LIN {X 0,Y 573.228,Z 217.081,A -85,B 0,C 180,E1 -2311.435,E2 -2311.435} C_VEL
LIN {X 0,Y 573.254,Z 217.075,A -85,B 0,C 180,E1 -2314.59,E2 -2314.59} C_VEL
LIN {X 0,Y 573.238,Z 217.078,A -85,B 0,C 180,E1 -2317.662,E2 -2317.662} C_VEL
LIN {X 0,Y 573.273,Z 217.079,A -85,B 0,C 180,E1 -2320.67,E2 -2320.67} C_VEL
LIN {X 0,Y 573.21,Z 217.081,A -85,B 0,C 180,E1 -2323.621,E2 -2323.621} C_VEL
LIN {X 0,Y 573.252,Z 217.08,A -85,B 0,C 180,E1 -2325.807,E2 -2325.807} C_VEL
LIN {X 0,Y 573.232,Z 217.077,A -85,B 0,C 180,E1 -2328.765,E2 -2328.765} C_VEL
LIN {X 0,Y 573.248,Z 217.08,A -85,B 0,C 180,E1 -2331.54,E2 -2331.54} C_VEL
LIN {X 0,Y 573.243,Z 217.077,A -85,B 0,C 180,E1 -2333.665,E2 -2333.665} C_VEL
LIN {X 0,Y 573.225,Z 217.079,A -85,B 0,C 180,E1 -2335.781,E2 -2335.781} C_VEL
LIN {X 0,Y 573.311,Z 217.07,A -85,B 0,C 180,E1 -2337.892,E2 -2337.892} C_VEL
LIN {X 0,Y 573.326,Z 217.067,A -85,B 0,C 180,E1 -2340.702,E2 -2340.702} C_VEL
LIN {X 0,Y 573.292,Z 217.07,A -85,B 0,C 180,E1 -2342.811,E2 -2342.811} C_VEL
LIN {X 0,Y 573.274,Z 217.077,A -85,B 0,C 180,E1 -2345.628,E2 -2345.628} C_VEL
LIN {X 0,Y 573.235,Z 217.078,A -85,B 0,C 180,E1 -2348.46,E2 -2348.46} C_VEL
LIN {X 0,Y 573.28,Z 217.073,A -85,B 0,C 180,E1 -2351.312,E2 -2351.312} C_VEL
LIN {X 0,Y 573.283,Z 217.078,A -85,B 0,C 180,E1 -2354.422,E2 -2354.422} C_VEL
LIN {X 0,Y 573.266,Z 217.074,A -85,B 0,C 180,E1 -2357.112,E2 -2357.112} C_VEL
LIN {X 0,Y 573.244,Z 217.078,A -85,B 0,C 180,E1 -2360.077,E2 -2360.077} C_VEL
LIN {X 0,Y 573.227,Z 217.078,A -85,B 0,C 180,E1 -2362.338,E2 -2362.338} C_VEL
LIN {X 0,Y 573.193,Z 217.083,A -85,B 0,C 180,E1 -2364.335,E2 -2364.335} C_VEL
LIN {X 0,Y 572.549,Z 217.17,A -85,B 0,C 180,E1 -2364.921,E2 -2364.921} C_VEL
LIN {X 0,Y 569.716,Z 217.52,A -85,B 0,C 180,E1 -2365.873,E2 -2365.873} C_VEL
LIN {X 0,Y 567.301,Z 217.822,A -85,B 0,C 180,E1 -2366.638,E2 -2366.638} C_VEL
LIN {X 0,Y 566.251,Z 217.949,A -85,B 0,C 180,E1 -2367.229,E2 -2367.229} C_VEL
LIN {X 0,Y 566.158,Z 217.958,A -85,B 0,C 180,E1 -2367.43,E2 -2367.43} C_VEL
LIN {X 0,Y 566.175,Z 217.958,A -85,B 0,C 180,E1 -2369.771,E2 -2369.771} C_VEL
LIN {X 0,Y 566.209,Z 217.956,A -85,B 0,C 180,E1 -2372.429,E2 -2372.429} C_VEL
LIN {X 0,Y 566.186,Z 217.956,A -85,B 0,C 180,E1 -2374.989,E2 -2374.989} C_VEL
LIN {X 0,Y 566.199,Z 217.96,A -85,B 0,C 180,E1 -2377.461,E2 -2377.461} C_VEL
LIN {X 0,Y 566.214,Z 217.952,A -85,B 0,C 180,E1 -2380.199,E2 -2380.199} C_VEL
LIN {X 0,Y 566.193,Z 217.958,A -85,B 0,C 180,E1 -2383.055,E2 -2383.055} C_VEL
LIN {X 0,Y 566.15,Z 217.964,A -85,B 0,C 180,E1 -2386.054,E2 -2386.054} C_VEL
LIN {X 0,Y 566.141,Z 217.96,A -85,B 0,C 180,E1 -2388.856,E2 -2388.856} C_VEL
LIN {X 0,Y 566.187,Z 217.963,A -85,B 0,C 180,E1 -2391.636,E2 -2391.636} C_VEL
LIN {X 0,Y 566.158,Z 217.959,A -85,B 0,C 180,E1 -2394.307,E2 -2394.307} C_VEL
LIN {X 0,Y 566.206,Z 217.959,A -85,B 0,C 180,E1 -2396.896,E2 -2396.896} C_VEL
LIN {X 0,Y 566.063,Z 217.978,A -85,B 0,C 180,E1 -2399.399,E2 -2399.399} C_VEL
LIN {X 0,Y 566.018,Z 219.482,A -85,B 0,C 180,E1 -2401.036,E2 -2401.036} C_VEL
LIN {X 0,Y 565.984,Z 222.214,A -85,B 0,C 180,E1 -2403.446,E2 -2403.446} C_VEL
LIN {X 0,Y 565.96,Z 224.896,A -85,B 0,C 180,E1 -2405.807,E2 -2405.807} C_VEL
LIN {X 0,Y 565.943,Z 228.388,A -85,B 0,C 180,E1 -2408.891,E2 -2408.891} C_VEL
LIN {X 0,Y 565.917,Z 230.996,A -85,B 0,C 180,E1 -2411.161,E2 -2411.161} C_VEL
LIN {X 0,Y 565.897,Z 233.568,A -85,B 0,C 180,E1 -2413.402,E2 -2413.402} C_VEL
LIN {X 0,Y 565.876,Z 237.059,A -85,B 0,C 180,E1 -2416.35,E2 -2416.35} C_VEL
LIN {X 0,Y 565.887,Z 240.835,A -85,B 0,C 180,E1 -2419.263,E2 -2419.263} C_VEL
LIN {X 0,Y 565.847,Z 243.676,A -85,B 0,C 180,E1 -2421.427,E2 -2421.427} C_VEL
LIN {X 0,Y 566.921,Z 251.031,A -85,B 0,C 180,E1 -2421.623,E2 -2421.623} C_VEL
LIN {X 0,Y 566.792,Z 264.125,A -85,B 0,C 180,E1 -2422.025,E2 -2422.025} C_VEL
LIN {X 0,Y 566.713,Z 275.551,A -85,B 0,C 180,E1 -2422.517,E2 -2422.517} C_VEL
LIN {X 0,Y 566.463,Z 287.212,A -85,B 0,C 180,E1 -2423.168,E2 -2423.168} C_VEL
LIN {X 0,Y 566.41,Z 298.182,A -85,B 0,C 180,E1 -2423.945,E2 -2423.945} C_VEL
LIN {X 0,Y 566.23,Z 308.312,A -85,B 0,C 180,E1 -2424.836,E2 -2424.836} C_VEL
LIN {X 0,Y 566.159,Z 316.567,A -85,B 0,C 180,E1 -2425.728,E2 -2425.728} C_VEL
LIN {X 0,Y 566.083,Z 324.665,A -85,B 0,C 180,E1 -2426.796,E2 -2426.796} C_VEL
LIN {X 0,Y 565.912,Z 331.198,A -85,B 0,C 180,E1 -2427.864,E2 -2427.864} C_VEL
LIN {X 0,Y 565.961,Z 336.406,A -85,B 0,C 180,E1 -2428.932,E2 -2428.932} C_VEL
LIN {X 0,Y 565.872,Z 340.467,A -85,B 0,C 180,E1 -2429.999,E2 -2429.999} C_VEL
LIN {X 0,Y 565.846,Z 342.6,A -85,B 0,C 180,E1 -2430.711,E2 -2430.711} C_VEL
LIN {X 0,Y 565.847,Z 344.276,A -85,B 0,C 180,E1 -2431.422,E2 -2431.422} C_VEL
LIN {X 0,Y 565.873,Z 346.433,A -85,B 0,C 180,E1 -2432.847,E2 -2432.847} C_VEL
LIN {X 0,Y 565.911,Z 346.898,A -85,B 0,C 180,E1 -2433.559,E2 -2433.559} C_VEL
LIN {X 0,Y 565.911,Z 346.957,A -85,B 0,C 180,E1 -2434.272,E2 -2434.272} C_VEL
LIN {X 0,Y 565.898,Z 345.923,A -85,B 0,C 180,E1 -2435.701,E2 -2435.701} C_VEL
LIN {X 0,Y 565.918,Z 344.547,A -85,B 0,C 180,E1 -2436.533,E2 -2436.533} C_VEL
LIN {X 0,Y 565.902,Z 341.227,A -85,B 0,C 180,E1 -2437.851,E2 -2437.851} C_VEL
LIN {X 0,Y 565.93,Z 337.36,A -85,B 0,C 180,E1 -2438.929,E2 -2438.929} C_VEL
LIN {X 0,Y 565.978,Z 332.342,A -85,B 0,C 180,E1 -2440.01,E2 -2440.01} C_VEL
LIN {X 0,Y 566.048,Z 325.124,A -85,B 0,C 180,E1 -2441.227,E2 -2441.227} C_VEL
LIN {X 0,Y 566.158,Z 316.558,A -85,B 0,C 180,E1 -2442.364,E2 -2442.364} C_VEL
LIN {X 0,Y 566.247,Z 308.118,A -85,B 0,C 180,E1 -2443.273,E2 -2443.273} C_VEL
LIN {X 0,Y 566.372,Z 297.678,A -85,B 0,C 180,E1 -2444.185,E2 -2444.185} C_VEL
LIN {X 0,Y 566.493,Z 286.979,A -85,B 0,C 180,E1 -2444.936,E2 -2444.936} C_VEL
LIN {X 0,Y 566.655,Z 275.898,A -85,B 0,C 180,E1 -2445.556,E2 -2445.556} C_VEL
LIN {X 0,Y 566.771,Z 264.256,A -85,B 0,C 180,E1 -2446.061,E2 -2446.061} C_VEL
LIN {X 0,Y 566.882,Z 250.786,A -85,B 0,C 180,E1 -2446.474,E2 -2446.474} C_VEL
LIN {X 0,Y 565.905,Z 243.69,A -85,B 0,C 180,E1 -2446.651,E2 -2446.651} C_VEL
LIN {X 0,Y 565.849,Z 239.839,A -85,B 0,C 180,E1 -2449.592,E2 -2449.592} C_VEL
LIN {X 0,Y 565.836,Z 236.886,A -85,B 0,C 180,E1 -2451.876,E2 -2451.876} C_VEL
LIN {X 0,Y 565.892,Z 234.162,A -85,B 0,C 180,E1 -2454.193,E2 -2454.193} C_VEL
LIN {X 0,Y 565.953,Z 231.389,A -85,B 0,C 180,E1 -2456.607,E2 -2456.607} C_VEL
LIN {X 0,Y 566.002,Z 227.922,A -85,B 0,C 180,E1 -2459.635,E2 -2459.635} C_VEL
LIN {X 0,Y 566.007,Z 224.804,A -85,B 0,C 180,E1 -2462.398,E2 -2462.398} C_VEL
LIN {X 0,Y 566.02,Z 221.892,A -85,B 0,C 180,E1 -2464.966,E2 -2464.966} C_VEL
LIN {X 0,Y 566.031,Z 219.071,A -85,B 0,C 180,E1 -2467.472,E2 -2467.472} C_VEL
LIN {X 0,Y 566.035,Z 217.981,A -85,B 0,C 180,E1 -2468.535,E2 -2468.535} C_VEL
LIN {X 0,Y 566.202,Z 217.957,A -85,B 0,C 180,E1 -2470.785,E2 -2470.785} C_VEL
LIN {X 0,Y 566.196,Z 217.957,A -85,B 0,C 180,E1 -2473.053,E2 -2473.053} C_VEL
LIN {X 0,Y 566.187,Z 217.962,A -85,B 0,C 180,E1 -2476.048,E2 -2476.048} C_VEL
LIN {X 0,Y 566.195,Z 217.961,A -85,B 0,C 180,E1 -2479.214,E2 -2479.214} C_VEL
LIN {X 0,Y 566.181,Z 217.957,A -85,B 0,C 180,E1 -2481.636,E2 -2481.636} C_VEL
LIN {X 0,Y 566.205,Z 217.96,A -85,B 0,C 180,E1 -2484.311,E2 -2484.311} C_VEL
LIN {X 0,Y 566.195,Z 217.955,A -85,B 0,C 180,E1 -2486.896,E2 -2486.896} C_VEL
LIN {X 0,Y 566.162,Z 217.963,A -85,B 0,C 180,E1 -2489.406,E2 -2489.406} C_VEL
LIN {X 0,Y 566.219,Z 217.952,A -85,B 0,C 180,E1 -2491.858,E2 -2491.858} C_VEL
LIN {X 0,Y 566.217,Z 217.957,A -85,B 0,C 180,E1 -2494.251,E2 -2494.251} C_VEL
LIN {X 0,Y 566.181,Z 217.957,A -85,B 0,C 180,E1 -2496.713,E2 -2496.713} C_VEL
LIN {X 0,Y 566.193,Z 217.955,A -85,B 0,C 180,E1 -2499.662,E2 -2499.662} C_VEL
LIN {X 0,Y 566.188,Z 217.959,A -85,B 0,C 180,E1 -2502.668,E2 -2502.668} C_VEL
LIN {X 0,Y 566.224,Z 217.958,A -85,B 0,C 180,E1 -2505.626,E2 -2505.626} C_VEL
LIN {X 0,Y 566.231,Z 217.953,A -85,B 0,C 180,E1 -2508.671,E2 -2508.671} C_VEL
LIN {X 0,Y 566.213,Z 217.952,A -85,B 0,C 180,E1 -2511.434,E2 -2511.434} C_VEL
LIN {X 0,Y 566.264,Z 217.948,A -85,B 0,C 180,E1 -2514.302,E2 -2514.302} C_VEL
LIN {X 0,Y 566.262,Z 217.947,A -85,B 0,C 180,E1 -2517.866,E2 -2517.866} C_VEL
LIN {X 0,Y 566.289,Z 217.947,A -85,B 0,C 180,E1 -2520.711,E2 -2520.711} C_VEL
LIN {X 0,Y 566.262,Z 217.947,A -85,B 0,C 180,E1 -2522.846,E2 -2522.846} C_VEL
LIN {X 0,Y 566.254,Z 217.951,A -85,B 0,C 180,E1 -2525.698,E2 -2525.698} C_VEL
LIN {X 0,Y 566.221,Z 217.956,A -85,B 0,C 180,E1 -2528.566,E2 -2528.566} C_VEL
LIN {X 0,Y 566.229,Z 217.951,A -85,B 0,C 180,E1 -2531.455,E2 -2531.455} C_VEL
LIN {X 0,Y 566.223,Z 217.951,A -85,B 0,C 180,E1 -2534.507,E2 -2534.507} C_VEL
LIN {X 0,Y 566.195,Z 217.957,A -85,B 0,C 180,E1 -2537.332,E2 -2537.332} C_VEL
LIN {X 0,Y 566.2,Z 217.954,A -85,B 0,C 180,E1 -2539.581,E2 -2539.581} C_VEL
LIN {X 0,Y 566.172,Z 217.964,A -85,B 0,C 180,E1 -2541.863,E2 -2541.863} C_VEL
LIN {X 0,Y 566.207,Z 217.958,A -85,B 0,C 180,E1 -2545.031,E2 -2545.031} C_VEL
LIN {X 0,Y 566.218,Z 217.953,A -85,B 0,C 180,E1 -2547.339,E2 -2547.339} C_VEL
LIN {X 0,Y 566.217,Z 217.954,A -85,B 0,C 180,E1 -2549.768,E2 -2549.768} C_VEL
LIN {X 0,Y 566.189,Z 217.956,A -85,B 0,C 180,E1 -2552.43,E2 -2552.43} C_VEL
LIN {X 0,Y 566.171,Z 217.964,A -85,B 0,C 180,E1 -2554.99,E2 -2554.99} C_VEL
LIN {X 0,Y 566.188,Z 217.955,A -85,B 0,C 180,E1 -2557.462,E2 -2557.462} C_VEL
LIN {X 0,Y 566.219,Z 217.956,A -85,B 0,C 180,E1 -2560.198,E2 -2560.198} C_VEL
LIN {X 0,Y 566.183,Z 217.96,A -85,B 0,C 180,E1 -2563.056,E2 -2563.056} C_VEL
LIN {X 0,Y 566.191,Z 217.957,A -85,B 0,C 180,E1 -2566.05,E2 -2566.05} C_VEL
LIN {X 0,Y 566.207,Z 217.955,A -85,B 0,C 180,E1 -2568.865,E2 -2568.865} C_VEL
LIN {X 0,Y 566.183,Z 217.963,A -85,B 0,C 180,E1 -2571.638,E2 -2571.638} C_VEL
LIN {X 0,Y 566.233,Z 218.116,A -85,B 0,C 180,E1 -2573.046,E2 -2573.046} C_VEL
LIN {X 0,Y 566.78,Z 221.921,A -85,B 0,C 180,E1 -2574.354,E2 -2574.354} C_VEL
LIN {X 0,Y 566.801,Z 228.672,A -85,B 0,C 180,E1 -2576.555,E2 -2576.555} C_VEL
LIN {X 0,Y 566.686,Z 235.896,A -85,B 0,C 180,E1 -2578.841,E2 -2578.841} C_VEL
LIN {X 0,Y 566.54,Z 245.751,A -85,B 0,C 180,E1 -2581.877,E2 -2581.877} C_VEL
LIN {X 0,Y 566.44,Z 255.913,A -85,B 0,C 180,E1 -2584.923,E2 -2584.923} C_VEL
LIN {X 0,Y 566.32,Z 266.934,A -85,B 0,C 180,E1 -2588.144,E2 -2588.144} C_VEL
LIN {X 0,Y 566.182,Z 277.525,A -85,B 0,C 180,E1 -2591.173,E2 -2591.173} C_VEL
LIN {X 0,Y 566.108,Z 288.116,A -85,B 0,C 180,E1 -2594.151,E2 -2594.151} C_VEL
LIN {X 0,Y 566,Z 298.707,A -85,B 0,C 180,E1 -2597.086,E2 -2597.086} C_VEL
LIN {X 0,Y 565.997,Z 299.62,A -85,B 0,C 180,E1 -2597.328,E2 -2597.328} C_VEL
LIN {X 0,Y 566.925,Z 306.429,A -85,B 0,C 180,E1 -2597.472,E2 -2597.472} C_VEL
LIN {X 0,Y 566.818,Z 318.536,A -85,B 0,C 180,E1 -2597.787,E2 -2597.787} C_VEL
LIN {X 0,Y 566.699,Z 330.345,A -85,B 0,C 180,E1 -2598.23,E2 -2598.23} C_VEL
LIN {X 0,Y 566.548,Z 341.718,A -85,B 0,C 180,E1 -2598.795,E2 -2598.795} C_VEL
LIN {X 0,Y 566.421,Z 353.494,A -85,B 0,C 180,E1 -2599.546,E2 -2599.546} C_VEL
LIN {X 0,Y 566.3,Z 363.659,A -85,B 0,C 180,E1 -2600.356,E2 -2600.356} C_VEL
LIN {X 0,Y 566.165,Z 372.797,A -85,B 0,C 180,E1 -2601.255,E2 -2601.255} C_VEL
LIN {X 0,Y 566.079,Z 381.699,A -85,B 0,C 180,E1 -2602.331,E2 -2602.331} C_VEL
LIN {X 0,Y 565.966,Z 388.962,A -85,B 0,C 180,E1 -2603.423,E2 -2603.423} C_VEL
LIN {X 0,Y 566.004,Z 393.686,A -85,B 0,C 180,E1 -2604.3,E2 -2604.3} C_VEL
LIN {X 0,Y 565.933,Z 398.376,A -85,B 0,C 180,E1 -2605.371,E2 -2605.371} C_VEL
LIN {X 0,Y 565.926,Z 401.96,A -85,B 0,C 180,E1 -2606.441,E2 -2606.441} C_VEL
LIN {X 0,Y 565.877,Z 403.811,A -85,B 0,C 180,E1 -2607.154,E2 -2607.154} C_VEL
LIN {X 0,Y 565.841,Z 405.202,A -85,B 0,C 180,E1 -2607.866,E2 -2607.866} C_VEL
LIN {X 0,Y 565.841,Z 406.785,A -85,B 0,C 180,E1 -2609.289,E2 -2609.289} C_VEL
LIN {X 0,Y 565.839,Z 407,A -85,B 0,C 180,E1 -2610.001,E2 -2610.001} C_VEL
LIN {X 0,Y 565.846,Z 406.184,A -85,B 0,C 180,E1 -2611.424,E2 -2611.424} C_VEL
LIN {X 0,Y 565.841,Z 405.199,A -85,B 0,C 180,E1 -2612.136,E2 -2612.136} C_VEL
LIN {X 0,Y 565.878,Z 403.807,A -85,B 0,C 180,E1 -2612.849,E2 -2612.849} C_VEL
LIN {X 0,Y 565.926,Z 400.893,A -85,B 0,C 180,E1 -2613.917,E2 -2613.917} C_VEL
LIN {X 0,Y 565.878,Z 396.945,A -85,B 0,C 180,E1 -2614.988,E2 -2614.988} C_VEL
LIN {X 0,Y 566.002,Z 391.861,A -85,B 0,C 180,E1 -2616.06,E2 -2616.06} C_VEL
LIN {X 0,Y 566.041,Z 385.463,A -85,B 0,C 180,E1 -2617.133,E2 -2617.133} C_VEL
LIN {X 0,Y 566.133,Z 377.47,A -85,B 0,C 180,E1 -2618.209,E2 -2618.209} C_VEL
LIN {X 0,Y 566.229,Z 369.327,A -85,B 0,C 180,E1 -2619.106,E2 -2619.106} C_VEL
LIN {X 0,Y 566.336,Z 359.39,A -85,B 0,C 180,E1 -2620.006,E2 -2620.006} C_VEL
LIN {X 0,Y 566.472,Z 348.314,A -85,B 0,C 180,E1 -2620.807,E2 -2620.807} C_VEL
LIN {X 0,Y 566.61,Z 335.932,A -85,B 0,C 180,E1 -2621.511,E2 -2621.511} C_VEL
LIN {X 0,Y 566.739,Z 323.739,A -85,B 0,C 180,E1 -2622.035,E2 -2622.035} C_VEL
LIN {X 0,Y 566.923,Z 310.311,A -85,B 0,C 180,E1 -2622.44,E2 -2622.44} C_VEL
LIN {X 0,Y 566.62,Z 303.611,A -85,B 0,C 180,E1 -2622.591,E2 -2622.591} C_VEL
LIN {X 0,Y 565.988,Z 299.527,A -85,B 0,C 180,E1 -2622.688,E2 -2622.688} C_VEL
LIN {X 0,Y 566.086,Z 289.432,A -85,B 0,C 180,E1 -2625.482,E2 -2625.482} C_VEL
LIN {X 0,Y 566.16,Z 278.841,A -85,B 0,C 180,E1 -2628.455,E2 -2628.455} C_VEL
LIN {X 0,Y 566.248,Z 269.574,A -85,B 0,C 180,E1 -2631.097,E2 -2631.097} C_VEL
LIN {X 0,Y 566.366,Z 260.306,A -85,B 0,C 180,E1 -2633.785,E2 -2633.785} C_VEL
LIN {X 0,Y 566.489,Z 251.039,A -85,B 0,C 180,E1 -2636.528,E2 -2636.528} C_VEL
LIN {X 0,Y 566.571,Z 241.772,A -85,B 0,C 180,E1 -2639.34,E2 -2639.34} C_VEL
LIN {X 0,Y 566.752,Z 232.505,A -85,B 0,C 180,E1 -2642.224,E2 -2642.224} C_VEL
LIN {X 0,Y 566.84,Z 223.614,A -85,B 0,C 180,E1 -2645.084,E2 -2645.084} C_VEL
LIN {X 0,Y 566.303,Z 218.605,A -85,B 0,C 180,E1 -2646.785,E2 -2646.785} C_VEL
LIN {X 0,Y 566.181,Z 217.963,A -85,B 0,C 180,E1 -2647.016,E2 -2647.016} C_VEL
LIN {X 0,Y 566.214,Z 217.954,A -85,B 0,C 180,E1 -2649.685,E2 -2649.685} C_VEL
LIN {X 0,Y 566.193,Z 217.961,A -85,B 0,C 180,E1 -2652.09,E2 -2652.09} C_VEL
LIN {X 0,Y 566.18,Z 217.957,A -85,B 0,C 180,E1 -2655.036,E2 -2655.036} C_VEL
LIN {X 0,Y 566.196,Z 217.958,A -85,B 0,C 180,E1 -2657.911,E2 -2657.911} C_VEL
LIN {X 0,Y 566.217,Z 217.954,A -85,B 0,C 180,E1 -2660.726,E2 -2660.726} C_VEL
LIN {X 0,Y 566.185,Z 217.956,A -85,B 0,C 180,E1 -2663.429,E2 -2663.429} C_VEL
LIN {X 0,Y 566.201,Z 217.958,A -85,B 0,C 180,E1 -2666.269,E2 -2666.269} C_VEL
LIN {X 0,Y 566.189,Z 217.955,A -85,B 0,C 180,E1 -2668.925,E2 -2668.925} C_VEL
LIN {X 0,Y 566.194,Z 217.961,A -85,B 0,C 180,E1 -2671.856,E2 -2671.856} C_VEL
LIN {X 0,Y 566.215,Z 217.952,A -85,B 0,C 180,E1 -2674.251,E2 -2674.251} C_VEL
LIN {X 0,Y 566.175,Z 217.96,A -85,B 0,C 180,E1 -2676.72,E2 -2676.72} C_VEL
LIN {X 0,Y 566.211,Z 217.952,A -85,B 0,C 180,E1 -2679.663,E2 -2679.663} C_VEL
LIN {X 0,Y 566.176,Z 217.958,A -85,B 0,C 180,E1 -2681.921,E2 -2681.921} C_VEL
LIN {X 0,Y 566.185,Z 217.955,A -85,B 0,C 180,E1 -2684.89,E2 -2684.89} C_VEL
LIN {X 0,Y 566.173,Z 217.963,A -85,B 0,C 180,E1 -2687.818,E2 -2687.818} C_VEL
LIN {X 0,Y 566.151,Z 217.961,A -85,B 0,C 180,E1 -2689.992,E2 -2689.992} C_VEL
LIN {X 0,Y 566.245,Z 217.953,A -85,B 0,C 180,E1 -2692.87,E2 -2692.87} C_VEL
LIN {X 0,Y 566.283,Z 217.949,A -85,B 0,C 180,E1 -2695.016,E2 -2695.016} C_VEL
LIN {X 0,Y 566.283,Z 217.945,A -85,B 0,C 180,E1 -2697.866,E2 -2697.866} C_VEL
LIN {X 0,Y 566.298,Z 217.943,A -85,B 0,C 180,E1 -2700.711,E2 -2700.711} C_VEL
LIN {X 0,Y 566.261,Z 217.946,A -85,B 0,C 180,E1 -2702.846,E2 -2702.846} C_VEL
LIN {X 0,Y 566.239,Z 217.953,A -85,B 0,C 180,E1 -2705.699,E2 -2705.699} C_VEL
LIN {X 0,Y 566.191,Z 217.956,A -85,B 0,C 180,E1 -2708.566,E2 -2708.566} C_VEL
LIN {X 0,Y 566.25,Z 217.948,A -85,B 0,C 180,E1 -2711.454,E2 -2711.454} C_VEL
LIN {X 0,Y 566.237,Z 217.955,A -85,B 0,C 180,E1 -2714.504,E2 -2714.504} C_VEL
LIN {X 0,Y 566.206,Z 217.954,A -85,B 0,C 180,E1 -2717.332,E2 -2717.332} C_VEL
LIN {X 0,Y 566.211,Z 217.953,A -85,B 0,C 180,E1 -2720.337,E2 -2720.337} C_VEL
LIN {X 0,Y 566.171,Z 217.963,A -85,B 0,C 180,E1 -2723.279,E2 -2723.279} C_VEL
LIN {X 0,Y 566.173,Z 217.956,A -85,B 0,C 180,E1 -2725.751,E2 -2725.751} C_VEL
LIN {X 0,Y 566.158,Z 217.958,A -85,B 0,C 180,E1 -2727.43,E2 -2727.43} C_VEL
LIN {X 0,Y 565.475,Z 218.046,A -85,B 0,C 180,E1 -2728.023,E2 -2728.023} C_VEL
LIN {X 0,Y 562.623,Z 218.401,A -85,B 0,C 180,E1 -2728.988,E2 -2728.988} C_VEL
LIN {X 0,Y 560.23,Z 218.701,A -85,B 0,C 180,E1 -2729.764,E2 -2729.764} C_VEL
LIN {X 0,Y 559.212,Z 218.831,A -85,B 0,C 180,E1 -2730.362,E2 -2730.362} C_VEL
LIN {X 0,Y 559.133,Z 218.835,A -85,B 0,C 180,E1 -2730.565,E2 -2730.565} C_VEL
LIN {X 0,Y 559.159,Z 218.831,A -85,B 0,C 180,E1 -2732.715,E2 -2732.715} C_VEL
LIN {X 0,Y 559.131,Z 218.838,A -85,B 0,C 180,E1 -2735.324,E2 -2735.324} C_VEL
LIN {X 0,Y 559.137,Z 218.835,A -85,B 0,C 180,E1 -2738.018,E2 -2738.018} C_VEL
LIN {X 0,Y 559.161,Z 218.837,A -85,B 0,C 180,E1 -2740.812,E2 -2740.812} C_VEL
LIN {X 0,Y 559.116,Z 218.836,A -85,B 0,C 180,E1 -2743.737,E2 -2743.737} C_VEL
LIN {X 0,Y 559.097,Z 218.846,A -85,B 0,C 180,E1 -2746.261,E2 -2746.261} C_VEL
LIN {X 0,Y 559.1,Z 218.837,A -85,B 0,C 180,E1 -2748.957,E2 -2748.957} C_VEL
LIN {X 0,Y 559.177,Z 218.831,A -85,B 0,C 180,E1 -2751.192,E2 -2751.192} C_VEL
LIN {X 0,Y 559.129,Z 218.837,A -85,B 0,C 180,E1 -2753.787,E2 -2753.787} C_VEL
LIN {X 0,Y 559.154,Z 218.833,A -85,B 0,C 180,E1 -2756.423,E2 -2756.423} C_VEL
LIN {X 0,Y 559.098,Z 218.845,A -85,B 0,C 180,E1 -2758.976,E2 -2758.976} C_VEL
LIN {X 0,Y 558.987,Z 218.859,A -85,B 0,C 180,E1 -2759.806,E2 -2759.806} C_VEL
LIN {X 0,Y 558.915,Z 221.544,A -85,B 0,C 180,E1 -2762.273,E2 -2762.273} C_VEL
LIN {X 0,Y 558.926,Z 224.475,A -85,B 0,C 180,E1 -2764.869,E2 -2764.869} C_VEL
LIN {X 0,Y 558.866,Z 227.822,A -85,B 0,C 180,E1 -2767.835,E2 -2767.835} C_VEL
LIN {X 0,Y 558.838,Z 231.29,A -85,B 0,C 180,E1 -2770.914,E2 -2770.914} C_VEL
LIN {X 0,Y 558.837,Z 233.92,A -85,B 0,C 180,E1 -2773.186,E2 -2773.186} C_VEL
LIN {X 0,Y 558.793,Z 237.384,A -85,B 0,C 180,E1 -2776.174,E2 -2776.174} C_VEL
LIN {X 0,Y 558.823,Z 240.49,A -85,B 0,C 180,E1 -2778.804,E2 -2778.804} C_VEL
LIN {X 0,Y 558.75,Z 243.686,A -85,B 0,C 180,E1 -2781.272,E2 -2781.272} C_VEL
LIN {X 0,Y 560.012,Z 252.179,A -85,B 0,C 180,E1 -2781.497,E2 -2781.497} C_VEL
LIN {X 0,Y 559.861,Z 264.293,A -85,B 0,C 180,E1 -2781.88,E2 -2781.88} C_VEL
LIN {X 0,Y 559.721,Z 276.549,A -85,B 0,C 180,E1 -2782.423,E2 -2782.423} C_VEL
LIN {X 0,Y 559.481,Z 288.067,A -85,B 0,C 180,E1 -2783.086,E2 -2783.086} C_VEL
LIN {X 0,Y 559.385,Z 298.841,A -85,B 0,C 180,E1 -2783.869,E2 -2783.869} C_VEL
LIN {X 0,Y 559.191,Z 308.817,A -85,B 0,C 180,E1 -2784.771,E2 -2784.771} C_VEL
LIN {X 0,Y 559.118,Z 316.988,A -85,B 0,C 180,E1 -2785.674,E2 -2785.674} C_VEL
LIN {X 0,Y 559.029,Z 325.013,A -85,B 0,C 180,E1 -2786.756,E2 -2786.756} C_VEL
LIN {X 0,Y 558.824,Z 331.485,A -85,B 0,C 180,E1 -2787.837,E2 -2787.837} C_VEL
LIN {X 0,Y 558.886,Z 336.632,A -85,B 0,C 180,E1 -2788.918,E2 -2788.918} C_VEL
LIN {X 0,Y 558.775,Z 340.643,A -85,B 0,C 180,E1 -2789.999,E2 -2789.999} C_VEL
LIN {X 0,Y 558.747,Z 342.727,A -85,B 0,C 180,E1 -2790.72,E2 -2790.72} C_VEL
LIN {X 0,Y 558.747,Z 344.379,A -85,B 0,C 180,E1 -2791.44,E2 -2791.44} C_VEL
LIN {X 0,Y 558.794,Z 346.485,A -85,B 0,C 180,E1 -2792.883,E2 -2792.883} C_VEL
LIN {X 0,Y 558.82,Z 346.91,A -85,B 0,C 180,E1 -2793.604,E2 -2793.604} C_VEL
LIN {X 0,Y 558.762,Z 346.597,A -85,B 0,C 180,E1 -2795.05,E2 -2795.05} C_VEL
LIN {X 0,Y 558.81,Z 345.86,A -85,B 0,C 180,E1 -2795.773,E2 -2795.773} C_VEL
LIN {X 0,Y 558.846,Z 344.607,A -85,B 0,C 180,E1 -2796.534,E2 -2796.534} C_VEL
LIN {X 0,Y 558.829,Z 341.074,A -85,B 0,C 180,E1 -2797.951,E2 -2797.951} C_VEL
LIN {X 0,Y 558.833,Z 337.155,A -85,B 0,C 180,E1 -2799.043,E2 -2799.043} C_VEL
LIN {X 0,Y 558.903,Z 331.101,A -85,B 0,C 180,E1 -2800.321,E2 -2800.321} C_VEL
LIN {X 0,Y 558.997,Z 324.764,A -85,B 0,C 180,E1 -2801.371,E2 -2801.371} C_VEL
LIN {X 0,Y 559.112,Z 316.128,A -85,B 0,C 180,E1 -2802.522,E2 -2802.522} C_VEL
LIN {X 0,Y 559.201,Z 307.588,A -85,B 0,C 180,E1 -2803.444,E2 -2803.444} C_VEL
LIN {X 0,Y 559.355,Z 296.995,A -85,B 0,C 180,E1 -2804.367,E2 -2804.367} C_VEL
LIN {X 0,Y 559.513,Z 286.753,A -85,B 0,C 180,E1 -2805.088,E2 -2805.088} C_VEL
LIN {X 0,Y 559.717,Z 274.859,A -85,B 0,C 180,E1 -2805.754,E2 -2805.754} C_VEL
LIN {X 0,Y 559.826,Z 262.761,A -85,B 0,C 180,E1 -2806.265,E2 -2806.265} C_VEL
LIN {X 0,Y 559.905,Z 250.51,A -85,B 0,C 180,E1 -2806.638,E2 -2806.638} C_VEL
LIN {X 0,Y 558.777,Z 243.662,A -85,B 0,C 180,E1 -2806.836,E2 -2806.836} C_VEL
LIN {X 0,Y 558.749,Z 239.766,A -85,B 0,C 180,E1 -2809.852,E2 -2809.852} C_VEL
LIN {X 0,Y 558.765,Z 237.109,A -85,B 0,C 180,E1 -2812.167,E2 -2812.167} C_VEL
LIN {X 0,Y 558.836,Z 233.683,A -85,B 0,C 180,E1 -2815.111,E2 -2815.111} C_VEL
LIN {X 0,Y 558.863,Z 230.742,A -85,B 0,C 180,E1 -2817.728,E2 -2817.728} C_VEL
LIN {X 0,Y 558.903,Z 227.913,A -85,B 0,C 180,E1 -2820.196,E2 -2820.196} C_VEL
LIN {X 0,Y 558.918,Z 225.073,A -85,B 0,C 180,E1 -2822.729,E2 -2822.729} C_VEL
LIN {X 0,Y 558.946,Z 222.152,A -85,B 0,C 180,E1 -2825.336,E2 -2825.336} C_VEL
LIN {X 0,Y 558.978,Z 219.145,A -85,B 0,C 180,E1 -2828.028,E2 -2828.028} C_VEL
LIN {X 0,Y 559.141,Z 218.834,A -85,B 0,C 180,E1 -2829.939,E2 -2829.939} C_VEL
LIN {X 0,Y 559.156,Z 218.838,A -85,B 0,C 180,E1 -2832.742,E2 -2832.742} C_VEL
LIN {X 0,Y 559.144,Z 218.837,A -85,B 0,C 180,E1 -2835.76,E2 -2835.76} C_VEL
LIN {X 0,Y 559.152,Z 218.833,A -85,B 0,C 180,E1 -2838.228,E2 -2838.228} C_VEL
LIN {X 0,Y 559.168,Z 218.834,A -85,B 0,C 180,E1 -2841.19,E2 -2841.19} C_VEL
LIN {X 0,Y 559.166,Z 218.832,A -85,B 0,C 180,E1 -2843.791,E2 -2843.791} C_VEL
LIN {X 0,Y 559.139,Z 218.834,A -85,B 0,C 180,E1 -2846.423,E2 -2846.423} C_VEL
LIN {X 0,Y 559.14,Z 218.838,A -85,B 0,C 180,E1 -2848.979,E2 -2848.979} C_VEL
LIN {X 0,Y 559.186,Z 218.832,A -85,B 0,C 180,E1 -2852.288,E2 -2852.288} C_VEL
LIN {X 0,Y 559.17,Z 218.83,A -85,B 0,C 180,E1 -2854.812,E2 -2854.812} C_VEL
LIN {X 0,Y 559.128,Z 218.837,A -85,B 0,C 180,E1 -2857.846,E2 -2857.846} C_VEL
LIN {X 0,Y 559.181,Z 218.832,A -85,B 0,C 180,E1 -2860.494,E2 -2860.494} C_VEL
LIN {X 0,Y 559.172,Z 218.83,A -85,B 0,C 180,E1 -2863.197,E2 -2863.197} C_VEL
LIN {X 0,Y 559.164,Z 218.831,A -85,B 0,C 180,E1 -2866.184,E2 -2866.184} C_VEL
LIN {X 0,Y 559.186,Z 218.832,A -85,B 0,C 180,E1 -2869.133,E2 -2869.133} C_VEL
LIN {X 0,Y 559.193,Z 218.831,A -85,B 0,C 180,E1 -2872.053,E2 -2872.053} C_VEL
LIN {X 0,Y 559.255,Z 218.82,A -85,B 0,C 180,E1 -2874.953,E2 -2874.953} C_VEL
LIN {X 0,Y 559.235,Z 218.822,A -85,B 0,C 180,E1 -2877.839,E2 -2877.839} C_VEL
LIN {X 0,Y 559.259,Z 218.823,A -85,B 0,C 180,E1 -2880.72,E2 -2880.72} C_VEL
LIN {X 0,Y 559.229,Z 218.823,A -85,B 0,C 180,E1 -2882.881,E2 -2882.881} C_VEL
LIN {X 0,Y 559.223,Z 218.826,A -85,B 0,C 180,E1 -2885.77,E2 -2885.77} C_VEL
LIN {X 0,Y 559.179,Z 218.835,A -85,B 0,C 180,E1 -2888.674,E2 -2888.674} C_VEL
LIN {X 0,Y 559.193,Z 218.829,A -85,B 0,C 180,E1 -2891.601,E2 -2891.601} C_VEL
LIN {X 0,Y 559.188,Z 218.827,A -85,B 0,C 180,E1 -2894.596,E2 -2894.596} C_VEL
LIN {X 0,Y 559.154,Z 218.832,A -85,B 0,C 180,E1 -2897.557,E2 -2897.557} C_VEL
LIN {X 0,Y 559.16,Z 218.832,A -85,B 0,C 180,E1 -2899.838,E2 -2899.838} C_VEL
LIN {X 0,Y 559.121,Z 218.839,A -85,B 0,C 180,E1 -2902.154,E2 -2902.154} C_VEL
LIN {X 0,Y 559.169,Z 218.836,A -85,B 0,C 180,E1 -2905.299,E2 -2905.299} C_VEL
LIN {X 0,Y 559.186,Z 218.828,A -85,B 0,C 180,E1 -2907.712,E2 -2907.712} C_VEL
LIN {X 0,Y 559.155,Z 218.838,A -85,B 0,C 180,E1 -2910.183,E2 -2910.183} C_VEL
LIN {X 0,Y 559.145,Z 218.833,A -85,B 0,C 180,E1 -2912.716,E2 -2912.716} C_VEL
LIN {X 0,Y 559.118,Z 218.84,A -85,B 0,C 180,E1 -2915.325,E2 -2915.325} C_VEL
LIN {X 0,Y 559.127,Z 218.837,A -85,B 0,C 180,E1 -2918.018,E2 -2918.018} C_VEL
LIN {X 0,Y 559.164,Z 218.831,A -85,B 0,C 180,E1 -2920.812,E2 -2920.812} C_VEL
LIN {X 0,Y 559.127,Z 218.837,A -85,B 0,C 180,E1 -2923.735,E2 -2923.735} C_VEL
LIN {X 0,Y 559.14,Z 218.839,A -85,B 0,C 180,E1 -2926.804,E2 -2926.804} C_VEL
LIN {X 0,Y 559.171,Z 218.832,A -85,B 0,C 180,E1 -2929.191,E2 -2929.191} C_VEL
LIN {X 0,Y 559.128,Z 218.841,A -85,B 0,C 180,E1 -2931.984,E2 -2931.984} C_VEL
LIN {X 0,Y 559.194,Z 218.947,A -85,B 0,C 180,E1 -2932.799,E2 -2932.799} C_VEL
LIN {X 0,Y 559.834,Z 223.247,A -85,B 0,C 180,E1 -2934.287,E2 -2934.287} C_VEL
LIN {X 0,Y 559.853,Z 229.865,A -85,B 0,C 180,E1 -2936.474,E2 -2936.474} C_VEL
LIN {X 0,Y 559.696,Z 237.808,A -85,B 0,C 180,E1 -2939.015,E2 -2939.015} C_VEL
LIN {X 0,Y 559.527,Z 248.399,A -85,B 0,C 180,E1 -2942.308,E2 -2942.308} C_VEL
LIN {X 0,Y 559.414,Z 257.738,A -85,B 0,C 180,E1 -2945.134,E2 -2945.134} C_VEL
LIN {X 0,Y 559.291,Z 266.934,A -85,B 0,C 180,E1 -2947.855,E2 -2947.855} C_VEL
LIN {X 0,Y 559.175,Z 276.04,A -85,B 0,C 180,E1 -2950.5,E2 -2950.5} C_VEL
LIN {X 0,Y 559.05,Z 286.792,A -85,B 0,C 180,E1 -2953.571,E2 -2953.571} C_VEL
LIN {X 0,Y 558.961,Z 297.383,A -85,B 0,C 180,E1 -2956.551,E2 -2956.551} C_VEL
LIN {X 0,Y 558.941,Z 299.809,A -85,B 0,C 180,E1 -2957.169,E2 -2957.169} C_VEL
LIN {X 0,Y 560.015,Z 307.567,A -85,B 0,C 180,E1 -2957.338,E2 -2957.338} C_VEL
LIN {X 0,Y 559.881,Z 319.91,A -85,B 0,C 180,E1 -2957.68,E2 -2957.68} C_VEL
LIN {X 0,Y 559.729,Z 332.307,A -85,B 0,C 180,E1 -2958.172,E2 -2958.172} C_VEL
LIN {X 0,Y 559.54,Z 343.928,A -85,B 0,C 180,E1 -2958.782,E2 -2958.782} C_VEL
LIN {X 0,Y 559.432,Z 354.762,A -85,B 0,C 180,E1 -2959.506,E2 -2959.506} C_VEL
LIN {X 0,Y 559.243,Z 365.613,A -85,B 0,C 180,E1 -2960.416,E2 -2960.416} C_VEL
LIN {X 0,Y 559.126,Z 374.423,A -85,B 0,C 180,E1 -2961.326,E2 -2961.326} C_VEL
LIN {X 0,Y 558.995,Z 383.008,A -85,B 0,C 180,E1 -2962.415,E2 -2962.415} C_VEL
LIN {X 0,Y 558.884,Z 390.693,A -85,B 0,C 180,E1 -2963.65,E2 -2963.65} C_VEL
LIN {X 0,Y 558.869,Z 395.37,A -85,B 0,C 180,E1 -2964.589,E2 -2964.589} C_VEL
LIN {X 0,Y 558.868,Z 399.681,A -85,B 0,C 180,E1 -2965.674,E2 -2965.674} C_VEL
LIN {X 0,Y 558.836,Z 401.96,A -85,B 0,C 180,E1 -2966.396,E2 -2966.396} C_VEL
LIN {X 0,Y 558.799,Z 403.811,A -85,B 0,C 180,E1 -2967.117,E2 -2967.117} C_VEL
LIN {X 0,Y 558.746,Z 405.201,A -85,B 0,C 180,E1 -2967.839,E2 -2967.839} C_VEL
LIN {X 0,Y 558.741,Z 406.785,A -85,B 0,C 180,E1 -2969.28,E2 -2969.28} C_VEL
LIN {X 0,Y 558.74,Z 407,A -85,B 0,C 180,E1 -2970.001,E2 -2970.001} C_VEL
LIN {X 0,Y 558.745,Z 406.184,A -85,B 0,C 180,E1 -2971.443,E2 -2971.443} C_VEL
LIN {X 0,Y 558.747,Z 405.199,A -85,B 0,C 180,E1 -2972.164,E2 -2972.164} C_VEL
LIN {X 0,Y 558.799,Z 403.807,A -85,B 0,C 180,E1 -2972.885,E2 -2972.885} C_VEL
LIN {X 0,Y 558.844,Z 400.893,A -85,B 0,C 180,E1 -2973.967,E2 -2973.967} C_VEL
LIN {X 0,Y 558.798,Z 396.945,A -85,B 0,C 180,E1 -2975.052,E2 -2975.052} C_VEL
LIN {X 0,Y 558.922,Z 391.861,A -85,B 0,C 180,E1 -2976.137,E2 -2976.137} C_VEL
LIN {X 0,Y 558.978,Z 385.462,A -85,B 0,C 180,E1 -2977.224,E2 -2977.224} C_VEL
LIN {X 0,Y 559.097,Z 377.47,A -85,B 0,C 180,E1 -2978.313,E2 -2978.313} C_VEL
LIN {X 0,Y 559.195,Z 369.327,A -85,B 0,C 180,E1 -2979.222,E2 -2979.222} C_VEL
LIN {X 0,Y 559.336,Z 359.39,A -85,B 0,C 180,E1 -2980.133,E2 -2980.133} C_VEL
LIN {X 0,Y 559.477,Z 348.422,A -85,B 0,C 180,E1 -2980.936,E2 -2980.936} C_VEL
LIN {X 0,Y 559.638,Z 336.804,A -85,B 0,C 180,E1 -2981.611,E2 -2981.611} C_VEL
LIN {X 0,Y 559.778,Z 324.963,A -85,B 0,C 180,E1 -2982.14,E2 -2982.14} C_VEL
LIN {X 0,Y 559.978,Z 312.138,A -85,B 0,C 180,E1 -2982.55,E2 -2982.55} C_VEL
LIN {X 0,Y 559.803,Z 305.052,A -85,B 0,C 180,E1 -2982.718,E2 -2982.718} C_VEL
LIN {X 0,Y 558.934,Z 299.527,A -85,B 0,C 180,E1 -2982.851,E2 -2982.851} C_VEL
LIN {X 0,Y 559.05,Z 289.432,A -85,B 0,C 180,E1 -2985.682,E2 -2985.682} C_VEL
LIN {X 0,Y 559.13,Z 278.841,A -85,B 0,C 180,E1 -2988.696,E2 -2988.696} C_VEL
LIN {X 0,Y 559.229,Z 268.913,A -85,B 0,C 180,E1 -2991.568,E2 -2991.568} C_VEL
LIN {X 0,Y 559.388,Z 258.983,A -85,B 0,C 180,E1 -2994.495,E2 -2994.495} C_VEL
LIN {X 0,Y 559.52,Z 249.717,A -85,B 0,C 180,E1 -2997.289,E2 -2997.289} C_VEL
LIN {X 0,Y 559.648,Z 240.448,A -85,B 0,C 180,E1 -3000.154,E2 -3000.154} C_VEL
LIN {X 0,Y 559.777,Z 232.323,A -85,B 0,C 180,E1 -3002.734,E2 -3002.734} C_VEL
LIN {X 0,Y 559.876,Z 224.413,A -85,B 0,C 180,E1 -3005.32,E2 -3005.32} C_VEL
LIN {X 0,Y 559.544,Z 220.971,A -85,B 0,C 180,E1 -3006.5,E2 -3006.5} C_VEL
LIN {X 0,Y 559.156,Z 218.838,A -85,B 0,C 180,E1 -3007.303,E2 -3007.303} C_VEL
LIN {X 0,Y 559.162,Z 218.834,A -85,B 0,C 180,E1 -3009.942,E2 -3009.942} C_VEL
LIN {X 0,Y 559.161,Z 218.833,A -85,B 0,C 180,E1 -3012.745,E2 -3012.745} C_VEL
LIN {X 0,Y 559.16,Z 218.839,A -85,B 0,C 180,E1 -3015.761,E2 -3015.761} C_VEL
LIN {X 0,Y 559.169,Z 218.83,A -85,B 0,C 180,E1 -3018.23,E2 -3018.23} C_VEL
LIN {X 0,Y 559.178,Z 218.834,A -85,B 0,C 180,E1 -3021.193,E2 -3021.193} C_VEL
LIN {X 0,Y 559.122,Z 218.835,A -85,B 0,C 180,E1 -3023.788,E2 -3023.788} C_VEL
LIN {X 0,Y 559.142,Z 218.84,A -85,B 0,C 180,E1 -3026.424,E2 -3026.424} C_VEL
LIN {X 0,Y 559.154,Z 218.831,A -85,B 0,C 180,E1 -3028.98,E2 -3028.98} C_VEL
LIN {X 0,Y 559.139,Z 218.839,A -85,B 0,C 180,E1 -3031.626,E2 -3031.626} C_VEL
LIN {X 0,Y 559.179,Z 218.831,A -85,B 0,C 180,E1 -3033.903,E2 -3033.903} C_VEL
LIN {X 0,Y 559.144,Z 218.834,A -85,B 0,C 180,E1 -3036.572,E2 -3036.572} C_VEL
LIN {X 0,Y 559.181,Z 218.829,A -85,B 0,C 180,E1 -3039.396,E2 -3039.396} C_VEL
LIN {X 0,Y 559.127,Z 218.835,A -85,B 0,C 180,E1 -3041.685,E2 -3041.685} C_VEL
LIN {X 0,Y 559.134,Z 218.835,A -85,B 0,C 180,E1 -3044.695,E2 -3044.695} C_VEL
LIN {X 0,Y 559.143,Z 218.839,A -85,B 0,C 180,E1 -3047.662,E2 -3047.662} C_VEL
LIN {X 0,Y 559.112,Z 218.839,A -85,B 0,C 180,E1 -3049.864,E2 -3049.864} C_VEL
LIN {X 0,Y 559.207,Z 218.829,A -85,B 0,C 180,E1 -3052.78,E2 -3052.78} C_VEL
LIN {X 0,Y 559.257,Z 218.825,A -85,B 0,C 180,E1 -3054.953,E2 -3054.953} C_VEL
LIN {X 0,Y 559.255,Z 218.82,A -85,B 0,C 180,E1 -3057.84,E2 -3057.84} C_VEL
LIN {X 0,Y 559.269,Z 218.818,A -85,B 0,C 180,E1 -3060.72,E2 -3060.72} C_VEL
LIN {X 0,Y 559.229,Z 218.822,A -85,B 0,C 180,E1 -3062.882,E2 -3062.882} C_VEL
LIN {X 0,Y 559.206,Z 218.828,A -85,B 0,C 180,E1 -3065.771,E2 -3065.771} C_VEL
LIN {X 0,Y 559.158,Z 218.833,A -85,B 0,C 180,E1 -3068.675,E2 -3068.675} C_VEL
LIN {X 0,Y 559.212,Z 218.824,A -85,B 0,C 180,E1 -3071.6,E2 -3071.6} C_VEL
LIN {X 0,Y 559.209,Z 218.829,A -85,B 0,C 180,E1 -3074.595,E2 -3074.595} C_VEL
LIN {X 0,Y 559.149,Z 218.836,A -85,B 0,C 180,E1 -3077.557,E2 -3077.557} C_VEL
LIN {X 0,Y 559.172,Z 218.835,A -85,B 0,C 180,E1 -3079.838,E2 -3079.838} C_VEL
LIN {X 0,Y 559.138,Z 218.834,A -85,B 0,C 180,E1 -3082.153,E2 -3082.153} C_VEL
LIN {X 0,Y 559.123,Z 218.84,A -85,B 0,C 180,E1 -3085.173,E2 -3085.173} C_VEL
LIN {X 0,Y 559.112,Z 218.836,A -85,B 0,C 180,E1 -3087.716,E2 -3087.716} C_VEL
LIN {X 0,Y 559.133,Z 218.835,A -85,B 0,C 180,E1 -3090.565,E2 -3090.565} C_VEL
LIN {X 0,Y 558.476,Z 218.917,A -85,B 0,C 180,E1 -3091.167,E2 -3091.167} C_VEL
LIN {X 0,Y 555.619,Z 219.279,A -85,B 0,C 180,E1 -3092.143,E2 -3092.143} C_VEL
LIN {X 0,Y 553.204,Z 219.575,A -85,B 0,C 180,E1 -3092.928,E2 -3092.928} C_VEL
LIN {X 0,Y 552.175,Z 219.704,A -85,B 0,C 180,E1 -3093.535,E2 -3093.535} C_VEL
LIN {X 0,Y 552.096,Z 219.712,A -85,B 0,C 180,E1 -3093.741,E2 -3093.741} C_VEL
LIN {X 0,Y 552.106,Z 219.71,A -85,B 0,C 180,E1 -3096.747,E2 -3096.747} C_VEL
LIN {X 0,Y 552.135,Z 219.709,A -85,B 0,C 180,E1 -3099.527,E2 -3099.527} C_VEL
LIN {X 0,Y 552.116,Z 219.712,A -85,B 0,C 180,E1 -3102.427,E2 -3102.427} C_VEL
LIN {X 0,Y 552.072,Z 219.713,A -85,B 0,C 180,E1 -3105.559,E2 -3105.559} C_VEL
LIN {X 0,Y 552.057,Z 219.716,A -85,B 0,C 180,E1 -3108.547,E2 -3108.547} C_VEL
LIN {X 0,Y 552.12,Z 219.712,A -85,B 0,C 180,E1 -3111.41,E2 -3111.41} C_VEL
LIN {X 0,Y 552.083,Z 219.713,A -85,B 0,C 180,E1 -3114.155,E2 -3114.155} C_VEL
LIN {X 0,Y 552.112,Z 219.714,A -85,B 0,C 180,E1 -3116.813,E2 -3116.813} C_VEL
LIN {X 0,Y 552.006,Z 219.729,A -85,B 0,C 180,E1 -3119.384,E2 -3119.384} C_VEL
LIN {X 0,Y 551.919,Z 219.896,A -85,B 0,C 180,E1 -3120.223,E2 -3120.223} C_VEL
LIN {X 0,Y 551.857,Z 223.087,A -85,B 0,C 180,E1 -3123.058,E2 -3123.058} C_VEL
LIN {X 0,Y 551.834,Z 226.331,A -85,B 0,C 180,E1 -3125.948,E2 -3125.948} C_VEL
LIN {X 0,Y 551.779,Z 229.908,A -85,B 0,C 180,E1 -3129.105,E2 -3129.105} C_VEL
LIN {X 0,Y 551.735,Z 232.485,A -85,B 0,C 180,E1 -3131.43,E2 -3131.43} C_VEL
LIN {X 0,Y 551.731,Z 235.111,A -85,B 0,C 180,E1 -3133.725,E2 -3133.725} C_VEL
LIN {X 0,Y 551.716,Z 237.763,A -85,B 0,C 180,E1 -3135.993,E2 -3135.993} C_VEL
LIN {X 0,Y 551.739,Z 241.18,A -85,B 0,C 180,E1 -3138.984,E2 -3138.984} C_VEL
LIN {X 0,Y 551.689,Z 243.666,A -85,B 0,C 180,E1 -3141.09,E2 -3141.09} C_VEL
LIN {X 0,Y 553.072,Z 252.434,A -85,B 0,C 180,E1 -3141.343,E2 -3141.343} C_VEL
LIN {X 0,Y 552.933,Z 264.458,A -85,B 0,C 180,E1 -3141.732,E2 -3141.732} C_VEL
LIN {X 0,Y 552.791,Z 275.794,A -85,B 0,C 180,E1 -3142.236,E2 -3142.236} C_VEL
LIN {X 0,Y 552.512,Z 287.219,A -85,B 0,C 180,E1 -3142.89,E2 -3142.89} C_VEL
LIN {X 0,Y 552.383,Z 298.351,A -85,B 0,C 180,E1 -3143.699,E2 -3143.699} C_VEL
LIN {X 0,Y 552.213,Z 307.54,A -85,B 0,C 180,E1 -3144.522,E2 -3144.522} C_VEL
LIN {X 0,Y 552.094,Z 315.934,A -85,B 0,C 180,E1 -3145.436,E2 -3145.436} C_VEL
LIN {X 0,Y 551.943,Z 324.141,A -85,B 0,C 180,E1 -3146.531,E2 -3146.531} C_VEL
LIN {X 0,Y 551.86,Z 330.764,A -85,B 0,C 180,E1 -3147.627,E2 -3147.627} C_VEL
LIN {X 0,Y 551.789,Z 336.847,A -85,B 0,C 180,E1 -3148.904,E2 -3148.904} C_VEL
LIN {X 0,Y 551.678,Z 340.81,A -85,B 0,C 180,E1 -3149.999,E2 -3149.999} C_VEL
LIN {X 0,Y 551.648,Z 342.854,A -85,B 0,C 180,E1 -3150.729,E2 -3150.729} C_VEL
LIN {X 0,Y 551.646,Z 344.482,A -85,B 0,C 180,E1 -3151.459,E2 -3151.459} C_VEL
LIN {X 0,Y 551.655,Z 345.71,A -85,B 0,C 180,E1 -3152.189,E2 -3152.189} C_VEL
LIN {X 0,Y 551.718,Z 346.527,A -85,B 0,C 180,E1 -3152.92,E2 -3152.92} C_VEL
LIN {X 0,Y 551.731,Z 346.921,A -85,B 0,C 180,E1 -3153.651,E2 -3153.651} C_VEL
LIN {X 0,Y 551.68,Z 346.562,A -85,B 0,C 180,E1 -3155.115,E2 -3155.115} C_VEL
LIN {X 0,Y 551.729,Z 344.747,A -85,B 0,C 180,E1 -3156.495,E2 -3156.495} C_VEL
LIN {X 0,Y 551.73,Z 341.992,A -85,B 0,C 180,E1 -3157.685,E2 -3157.685} C_VEL
LIN {X 0,Y 551.762,Z 338.385,A -85,B 0,C 180,E1 -3158.791,E2 -3158.791} C_VEL
LIN {X 0,Y 551.823,Z 333.648,A -85,B 0,C 180,E1 -3159.899,E2 -3159.899} C_VEL
LIN {X 0,Y 551.928,Z 327.633,A -85,B 0,C 180,E1 -3161.01,E2 -3161.01} C_VEL
LIN {X 0,Y 551.999,Z 320.115,A -85,B 0,C 180,E1 -3162.126,E2 -3162.126} C_VEL
LIN {X 0,Y 552.127,Z 312.423,A -85,B 0,C 180,E1 -3163.057,E2 -3163.057} C_VEL
LIN {X 0,Y 552.313,Z 303.055,A -85,B 0,C 180,E1 -3163.99,E2 -3163.99} C_VEL
LIN {X 0,Y 552.432,Z 293.194,A -85,B 0,C 180,E1 -3164.789,E2 -3164.789} C_VEL
LIN {X 0,Y 552.583,Z 282.503,A -85,B 0,C 180,E1 -3165.49,E2 -3165.49} C_VEL
LIN {X 0,Y 552.805,Z 270.699,A -85,B 0,C 180,E1 -3166.098,E2 -3166.098} C_VEL
LIN {X 0,Y 552.972,Z 258.556,A -85,B 0,C 180,E1 -3166.568,E2 -3166.568} C_VEL
LIN {X 0,Y 552.843,Z 250.673,A -85,B 0,C 180,E1 -3166.797,E2 -3166.797} C_VEL
LIN {X 0,Y 551.677,Z 243.68,A -85,B 0,C 180,E1 -3166.989,E2 -3166.989} C_VEL
LIN {X 0,Y 551.69,Z 240.038,A -85,B 0,C 180,E1 -3170.117,E2 -3170.117} C_VEL
LIN {X 0,Y 551.703,Z 237.425,A -85,B 0,C 180,E1 -3172.466,E2 -3172.466} C_VEL
LIN {X 0,Y 551.768,Z 234.122,A -85,B 0,C 180,E1 -3175.264,E2 -3175.264} C_VEL
LIN {X 0,Y 551.815,Z 230.896,A -85,B 0,C 180,E1 -3178.113,E2 -3178.113} C_VEL
LIN {X 0,Y 551.845,Z 228.068,A -85,B 0,C 180,E1 -3180.624,E2 -3180.624} C_VEL
LIN {X 0,Y 551.862,Z 225.198,A -85,B 0,C 180,E1 -3183.202,E2 -3183.202} C_VEL
LIN {X 0,Y 551.873,Z 222.26,A -85,B 0,C 180,E1 -3185.858,E2 -3185.858} C_VEL
LIN {X 0,Y 551.919,Z 220.038,A -85,B 0,C 180,E1 -3187.861,E2 -3187.861} C_VEL
LIN {X 0,Y 552.052,Z 219.722,A -85,B 0,C 180,E1 -3189.532,E2 -3189.532} C_VEL
LIN {X 0,Y 552.126,Z 219.71,A -85,B 0,C 180,E1 -3192.414,E2 -3192.414} C_VEL
LIN {X 0,Y 552.089,Z 219.714,A -85,B 0,C 180,E1 -3195.561,E2 -3195.561} C_VEL
LIN {X 0,Y 552.101,Z 219.711,A -85,B 0,C 180,E1 -3198.679,E2 -3198.679} C_VEL
LIN {X 0,Y 552.111,Z 219.711,A -85,B 0,C 180,E1 -3201.41,E2 -3201.41} C_VEL
LIN {X 0,Y 552.106,Z 219.715,A -85,B 0,C 180,E1 -3204.158,E2 -3204.158} C_VEL
LIN {X 0,Y 552.098,Z 219.711,A -85,B 0,C 180,E1 -3206.813,E2 -3206.813} C_VEL
LIN {X 0,Y 552.088,Z 219.716,A -85,B 0,C 180,E1 -3209.39,E2 -3209.39} C_VEL
LIN {X 0,Y 552.117,Z 219.709,A -85,B 0,C 180,E1 -3211.902,E2 -3211.902} C_VEL
LIN {X 0,Y 552.148,Z 219.706,A -85,B 0,C 180,E1 -3214.648,E2 -3214.648} C_VEL
LIN {X 0,Y 552.083,Z 219.718,A -85,B 0,C 180,E1 -3217.548,E2 -3217.548} C_VEL
LIN {X 0,Y 552.133,Z 219.709,A -85,B 0,C 180,E1 -3220.374,E2 -3220.374} C_VEL
LIN {X 0,Y 552.145,Z 219.705,A -85,B 0,C 180,E1 -3222.977,E2 -3222.977} C_VEL
LIN {X 0,Y 552.127,Z 219.709,A -85,B 0,C 180,E1 -3226.004,E2 -3226.004} C_VEL
LIN {X 0,Y 552.154,Z 219.71,A -85,B 0,C 180,E1 -3228.993,E2 -3228.993} C_VEL
LIN {X 0,Y 552.147,Z 219.708,A -85,B 0,C 180,E1 -3231.951,E2 -3231.951} C_VEL
LIN {X 0,Y 552.229,Z 219.695,A -85,B 0,C 180,E1 -3234.889,E2 -3234.889} C_VEL
LIN {X 0,Y 552.207,Z 219.698,A -85,B 0,C 180,E1 -3237.812,E2 -3237.812} C_VEL
LIN {X 0,Y 552.229,Z 219.698,A -85,B 0,C 180,E1 -3240.729,E2 -3240.729} C_VEL
LIN {X 0,Y 552.195,Z 219.699,A -85,B 0,C 180,E1 -3242.918,E2 -3242.918} C_VEL
LIN {X 0,Y 552.193,Z 219.701,A -85,B 0,C 180,E1 -3245.844,E2 -3245.844} C_VEL
LIN {X 0,Y 552.149,Z 219.71,A -85,B 0,C 180,E1 -3248.786,E2 -3248.786} C_VEL
LIN {X 0,Y 552.15,Z 219.708,A -85,B 0,C 180,E1 -3251.751,E2 -3251.751} C_VEL
LIN {X 0,Y 552.126,Z 219.708,A -85,B 0,C 180,E1 -3254.749,E2 -3254.749} C_VEL
LIN {X 0,Y 552.106,Z 219.71,A -85,B 0,C 180,E1 -3257.789,E2 -3257.789} C_VEL
LIN {X 0,Y 552.119,Z 219.712,A -85,B 0,C 180,E1 -3260.102,E2 -3260.102} C_VEL
LIN {X 0,Y 552.073,Z 219.715,A -85,B 0,C 180,E1 -3262.452,E2 -3262.452} C_VEL
LIN {X 0,Y 552.147,Z 219.709,A -85,B 0,C 180,E1 -3265.352,E2 -3265.352} C_VEL
LIN {X 0,Y 552.119,Z 219.71,A -85,B 0,C 180,E1 -3268.098,E2 -3268.098} C_VEL
LIN {X 0,Y 552.098,Z 219.712,A -85,B 0,C 180,E1 -3270.61,E2 -3270.61} C_VEL
LIN {X 0,Y 552.105,Z 219.714,A -85,B 0,C 180,E1 -3273.187,E2 -3273.187} C_VEL
LIN {X 0,Y 552.077,Z 219.714,A -85,B 0,C 180,E1 -3275.844,E2 -3275.844} C_VEL
LIN {X 0,Y 552.118,Z 219.709,A -85,B 0,C 180,E1 -3279.063,E2 -3279.063} C_VEL
LIN {X 0,Y 552.117,Z 219.713,A -85,B 0,C 180,E1 -3281.446,E2 -3281.446} C_VEL
LIN {X 0,Y 552.083,Z 219.715,A -85,B 0,C 180,E1 -3284.532,E2 -3284.532} C_VEL
LIN {X 0,Y 552.125,Z 219.709,A -85,B 0,C 180,E1 -3287.586,E2 -3287.586} C_VEL
LIN {X 0,Y 552.129,Z 219.711,A -85,B 0,C 180,E1 -3290.474,E2 -3290.474} C_VEL
LIN {X 0,Y 552.131,Z 219.862,A -85,B 0,C 180,E1 -3292.571,E2 -3292.571} C_VEL
LIN {X 0,Y 552.904,Z 225.191,A -85,B 0,C 180,E1 -3294.44,E2 -3294.44} C_VEL
LIN {X 0,Y 552.844,Z 233.037,A -85,B 0,C 180,E1 -3297.037,E2 -3297.037} C_VEL
LIN {X 0,Y 552.66,Z 241.793,A -85,B 0,C 180,E1 -3299.853,E2 -3299.853} C_VEL
LIN {X 0,Y 552.515,Z 251.615,A -85,B 0,C 180,E1 -3302.924,E2 -3302.924} C_VEL
LIN {X 0,Y 552.352,Z 261.638,A -85,B 0,C 180,E1 -3305.975,E2 -3305.975} C_VEL
LIN {X 0,Y 552.197,Z 270.905,A -85,B 0,C 180,E1 -3308.733,E2 -3308.733} C_VEL
LIN {X 0,Y 552.082,Z 280.173,A -85,B 0,C 180,E1 -3311.444,E2 -3311.444} C_VEL
LIN {X 0,Y 551.975,Z 290.764,A -85,B 0,C 180,E1 -3314.493,E2 -3314.493} C_VEL
LIN {X 0,Y 551.886,Z 299.534,A -85,B 0,C 180,E1 -3316.984,E2 -3316.984} C_VEL
LIN {X 0,Y 553.097,Z 308.569,A -85,B 0,C 180,E1 -3317.2,E2 -3317.2} C_VEL
LIN {X 0,Y 552.957,Z 321.21,A -85,B 0,C 180,E1 -3317.57,E2 -3317.57} C_VEL
LIN {X 0,Y 552.748,Z 333.51,A -85,B 0,C 180,E1 -3318.077,E2 -3318.077} C_VEL
LIN {X 0,Y 552.558,Z 345.401,A -85,B 0,C 180,E1 -3318.728,E2 -3318.728} C_VEL
LIN {X 0,Y 552.384,Z 357.111,A -85,B 0,C 180,E1 -3319.555,E2 -3319.555} C_VEL
LIN {X 0,Y 552.2,Z 367.55,A -85,B 0,C 180,E1 -3320.478,E2 -3320.478} C_VEL
LIN {X 0,Y 552.081,Z 375.999,A -85,B 0,C 180,E1 -3321.399,E2 -3321.399} C_VEL
LIN {X 0,Y 551.925,Z 384.245,A -85,B 0,C 180,E1 -3322.502,E2 -3322.502} C_VEL
LIN {X 0,Y 551.82,Z 391.213,A -85,B 0,C 180,E1 -3323.663,E2 -3323.663} C_VEL
LIN {X 0,Y 551.723,Z 396.954,A -85,B 0,C 180,E1 -3324.885,E2 -3324.885} C_VEL
LIN {X 0,Y 551.763,Z 400.899,A -85,B 0,C 180,E1 -3325.984,E2 -3325.984} C_VEL
LIN {X 0,Y 551.723,Z 403.811,A -85,B 0,C 180,E1 -3327.08,E2 -3327.08} C_VEL
LIN {X 0,Y 551.645,Z 406.187,A -85,B 0,C 180,E1 -3328.541,E2 -3328.541} C_VEL
LIN {X 0,Y 551.64,Z 407,A -85,B 0,C 180,E1 -3330.001,E2 -3330.001} C_VEL
LIN {X 0,Y 551.645,Z 406.185,A -85,B 0,C 180,E1 -3331.461,E2 -3331.461} C_VEL
LIN {X 0,Y 551.657,Z 405.198,A -85,B 0,C 180,E1 -3332.191,E2 -3332.191} C_VEL
LIN {X 0,Y 551.724,Z 403.807,A -85,B 0,C 180,E1 -3332.922,E2 -3332.922} C_VEL
LIN {X 0,Y 551.764,Z 400.893,A -85,B 0,C 180,E1 -3334.018,E2 -3334.018} C_VEL
LIN {X 0,Y 551.724,Z 396.945,A -85,B 0,C 180,E1 -3335.117,E2 -3335.117} C_VEL
LIN {X 0,Y 551.825,Z 391.188,A -85,B 0,C 180,E1 -3336.342,E2 -3336.342} C_VEL
LIN {X 0,Y 551.927,Z 384.23,A -85,B 0,C 180,E1 -3337.501,E2 -3337.501} C_VEL
LIN {X 0,Y 552.079,Z 375.982,A -85,B 0,C 180,E1 -3338.604,E2 -3338.604} C_VEL
LIN {X 0,Y 552.201,Z 367.527,A -85,B 0,C 180,E1 -3339.525,E2 -3339.525} C_VEL
LIN {X 0,Y 552.386,Z 357.084,A -85,B 0,C 180,E1 -3340.447,E2 -3340.447} C_VEL
LIN {X 0,Y 552.566,Z 345.335,A -85,B 0,C 180,E1 -3341.276,E2 -3341.276} C_VEL
LIN {X 0,Y 552.736,Z 333.463,A -85,B 0,C 180,E1 -3341.925,E2 -3341.925} C_VEL
LIN {X 0,Y 552.915,Z 321.145,A -85,B 0,C 180,E1 -3342.434,E2 -3342.434} C_VEL
LIN {X 0,Y 553.098,Z 308.48,A -85,B 0,C 180,E1 -3342.802,E2 -3342.802} C_VEL
LIN {X 0,Y 551.884,Z 299.527,A -85,B 0,C 180,E1 -3343.018,E2 -3343.018} C_VEL
LIN {X 0,Y 551.991,Z 289.432,A -85,B 0,C 180,E1 -3345.888,E2 -3345.888} C_VEL
LIN {X 0,Y 552.083,Z 278.841,A -85,B 0,C 180,E1 -3348.943,E2 -3348.943} C_VEL
LIN {X 0,Y 552.256,Z 268.251,A -85,B 0,C 180,E1 -3352.051,E2 -3352.051} C_VEL
LIN {X 0,Y 552.383,Z 258.983,A -85,B 0,C 180,E1 -3354.827,E2 -3354.827} C_VEL
LIN {X 0,Y 552.533,Z 249.715,A -85,B 0,C 180,E1 -3357.664,E2 -3357.664} C_VEL
LIN {X 0,Y 552.683,Z 240.448,A -85,B 0,C 180,E1 -3360.575,E2 -3360.575} C_VEL
LIN {X 0,Y 552.857,Z 232.505,A -85,B 0,C 180,E1 -3363.137,E2 -3363.137} C_VEL
LIN {X 0,Y 552.916,Z 225.215,A -85,B 0,C 180,E1 -3365.561,E2 -3365.561} C_VEL
LIN {X 0,Y 552.12,Z 219.714,A -85,B 0,C 180,E1 -3367.49,E2 -3367.49} C_VEL
LIN {X 0,Y 552.113,Z 219.716,A -85,B 0,C 180,E1 -3370.482,E2 -3370.482} C_VEL
LIN {X 0,Y 552.113,Z 219.71,A -85,B 0,C 180,E1 -3373.424,E2 -3373.424} C_VEL
LIN {X 0,Y 552.113,Z 219.709,A -85,B 0,C 180,E1 -3376.577,E2 -3376.577} C_VEL
LIN {X 0,Y 552.114,Z 219.714,A -85,B 0,C 180,E1 -3379.519,E2 -3379.519} C_VEL
LIN {X 0,Y 552.093,Z 219.712,A -85,B 0,C 180,E1 -3382.336,E2 -3382.336} C_VEL
LIN {X 0,Y 552.077,Z 219.715,A -85,B 0,C 180,E1 -3385.05,E2 -3385.05} C_VEL
LIN {X 0,Y 552.106,Z 219.71,A -85,B 0,C 180,E1 -3387.681,E2 -3387.681} C_VEL
LIN {X 0,Y 552.092,Z 219.716,A -85,B 0,C 180,E1 -3390.234,E2 -3390.234} C_VEL
LIN {X 0,Y 552.135,Z 219.707,A -85,B 0,C 180,E1 -3393.002,E2 -3393.002} C_VEL
LIN {X 0,Y 552.12,Z 219.714,A -85,B 0,C 180,E1 -3395.162,E2 -3395.162} C_VEL
LIN {X 0,Y 552.133,Z 219.708,A -85,B 0,C 180,E1 -3398.338,E2 -3398.338} C_VEL
LIN {X 0,Y 552.156,Z 219.709,A -85,B 0,C 180,E1 -3400.674,E2 -3400.674} C_VEL
LIN {X 0,Y 552.077,Z 219.715,A -85,B 0,C 180,E1 -3403.736,E2 -3403.736} C_VEL
LIN {X 0,Y 552.109,Z 219.716,A -85,B 0,C 180,E1 -3406.004,E2 -3406.004} C_VEL
LIN {X 0,Y 552.127,Z 219.708,A -85,B 0,C 180,E1 -3408.993,E2 -3408.993} C_VEL
LIN {X 0,Y 552.143,Z 219.706,A -85,B 0,C 180,E1 -3411.951,E2 -3411.951} C_VEL
LIN {X 0,Y 552.232,Z 219.7,A -85,B 0,C 180,E1 -3414.889,E2 -3414.889} C_VEL
LIN {X 0,Y 552.227,Z 219.696,A -85,B 0,C 180,E1 -3417.812,E2 -3417.812} C_VEL
LIN {X 0,Y 552.241,Z 219.694,A -85,B 0,C 180,E1 -3420.729,E2 -3420.729} C_VEL
LIN {X 0,Y 552.197,Z 219.698,A -85,B 0,C 180,E1 -3422.918,E2 -3422.918} C_VEL
LIN {X 0,Y 552.175,Z 219.703,A -85,B 0,C 180,E1 -3425.844,E2 -3425.844} C_VEL
LIN {X 0,Y 552.132,Z 219.71,A -85,B 0,C 180,E1 -3428.786,E2 -3428.786} C_VEL
LIN {X 0,Y 552.169,Z 219.702,A -85,B 0,C 180,E1 -3431.751,E2 -3431.751} C_VEL
LIN {X 0,Y 552.144,Z 219.707,A -85,B 0,C 180,E1 -3434.748,E2 -3434.748} C_VEL
LIN {X 0,Y 552.106,Z 219.716,A -85,B 0,C 180,E1 -3437.789,E2 -3437.789} C_VEL
LIN {X 0,Y 552.133,Z 219.708,A -85,B 0,C 180,E1 -3440.101,E2 -3440.101} C_VEL
LIN {X 0,Y 552.09,Z 219.712,A -85,B 0,C 180,E1 -3442.451,E2 -3442.451} C_VEL
LIN {X 0,Y 552.068,Z 219.717,A -85,B 0,C 180,E1 -3445.329,E2 -3445.329} C_VEL
LIN {X 0,Y 552.063,Z 219.716,A -85,B 0,C 180,E1 -3448.101,E2 -3448.101} C_VEL
LIN {X 0,Y 552.099,Z 219.714,A -85,B 0,C 180,E1 -3450.61,E2 -3450.61} C_VEL
LIN {X 0,Y 552.114,Z 219.709,A -85,B 0,C 180,E1 -3453.186,E2 -3453.186} C_VEL
LIN {X 0,Y 552.096,Z 219.712,A -85,B 0,C 180,E1 -3453.741,E2 -3453.741} C_VEL
LIN {X 0,Y 551.454,Z 219.795,A -85,B 0,C 180,E1 -3454.349,E2 -3454.349} C_VEL
LIN {X 0,Y 548.642,Z 220.145,A -85,B 0,C 180,E1 -3455.338,E2 -3455.338} C_VEL
LIN {X 0,Y 546.235,Z 220.443,A -85,B 0,C 180,E1 -3456.133,E2 -3456.133} C_VEL
LIN {X 0,Y 545.171,Z 220.575,A -85,B 0,C 180,E1 -3456.747,E2 -3456.747} C_VEL
LIN {X 0,Y 545.069,Z 220.588,A -85,B 0,C 180,E1 -3456.955,E2 -3456.955} C_VEL
LIN {X 0,Y 545.072,Z 220.586,A -85,B 0,C 180,E1 -3460.142,E2 -3460.142} C_VEL
LIN {X 0,Y 545.046,Z 220.595,A -85,B 0,C 180,E1 -3462.694,E2 -3462.694} C_VEL
LIN {X 0,Y 545.022,Z 220.592,A -85,B 0,C 180,E1 -3465.172,E2 -3465.172} C_VEL
LIN {X 0,Y 545.026,Z 220.593,A -85,B 0,C 180,E1 -3468.409,E2 -3468.409} C_VEL
LIN {X 0,Y 545.073,Z 220.585,A -85,B 0,C 180,E1 -3470.817,E2 -3470.817} C_VEL
LIN {X 0,Y 545.042,Z 220.594,A -85,B 0,C 180,E1 -3473.619,E2 -3473.619} C_VEL
LIN {X 0,Y 545.056,Z 220.589,A -85,B 0,C 180,E1 -3476.326,E2 -3476.326} C_VEL
LIN {X 0,Y 544.993,Z 220.602,A -85,B 0,C 180,E1 -3478.946,E2 -3478.946} C_VEL
LIN {X 0,Y 544.923,Z 220.611,A -85,B 0,C 180,E1 -3479.801,E2 -3479.801} C_VEL
LIN {X 0,Y 544.844,Z 221.05,A -85,B 0,C 180,E1 -3480.647,E2 -3480.647} C_VEL
LIN {X 0,Y 544.8,Z 223.853,A -85,B 0,C 180,E1 -3483.159,E2 -3483.159} C_VEL
LIN {X 0,Y 544.774,Z 226.603,A -85,B 0,C 180,E1 -3485.617,E2 -3485.617} C_VEL
LIN {X 0,Y 544.715,Z 230.206,A -85,B 0,C 180,E1 -3488.821,E2 -3488.821} C_VEL
LIN {X 0,Y 544.67,Z 232.861,A -85,B 0,C 180,E1 -3491.18,E2 -3491.18} C_VEL
LIN {X 0,Y 544.687,Z 235.475,A -85,B 0,C 180,E1 -3493.508,E2 -3493.508} C_VEL
LIN {X 0,Y 544.651,Z 238.119,A -85,B 0,C 180,E1 -3495.807,E2 -3495.807} C_VEL
LIN {X 0,Y 544.689,Z 241.614,A -85,B 0,C 180,E1 -3498.839,E2 -3498.839} C_VEL
LIN {X 0,Y 544.609,Z 244.004,A -85,B 0,C 180,E1 -3500.927,E2 -3500.927} C_VEL
LIN {X 0,Y 546.127,Z 253.798,A -85,B 0,C 180,E1 -3501.209,E2 -3501.209} C_VEL
LIN {X 0,Y 545.971,Z 265.941,A -85,B 0,C 180,E1 -3501.626,E2 -3501.626} C_VEL
LIN {X 0,Y 545.769,Z 278.684,A -85,B 0,C 180,E1 -3502.228,E2 -3502.228} C_VEL
LIN {X 0,Y 545.516,Z 289.929,A -85,B 0,C 180,E1 -3502.92,E2 -3502.92} C_VEL
LIN {X 0,Y 545.364,Z 300.081,A -85,B 0,C 180,E1 -3503.71,E2 -3503.71} C_VEL
LIN {X 0,Y 545.123,Z 309.826,A -85,B 0,C 180,E1 -3504.636,E2 -3504.636} C_VEL
LIN {X 0,Y 544.962,Z 319.291,A -85,B 0,C 180,E1 -3505.746,E2 -3505.746} C_VEL
LIN {X 0,Y 544.822,Z 326.841,A -85,B 0,C 180,E1 -3506.856,E2 -3506.856} C_VEL
LIN {X 0,Y 544.713,Z 333.824,A -85,B 0,C 180,E1 -3508.151,E2 -3508.151} C_VEL
LIN {X 0,Y 544.577,Z 338.473,A -85,B 0,C 180,E1 -3509.259,E2 -3509.259} C_VEL
LIN {X 0,Y 544.639,Z 342.026,A -85,B 0,C 180,E1 -3510.369,E2 -3510.369} C_VEL
LIN {X 0,Y 544.547,Z 344.584,A -85,B 0,C 180,E1 -3511.478,E2 -3511.478} C_VEL
LIN {X 0,Y 544.57,Z 345.788,A -85,B 0,C 180,E1 -3512.218,E2 -3512.218} C_VEL
LIN {X 0,Y 544.645,Z 346.56,A -85,B 0,C 180,E1 -3512.958,E2 -3512.958} C_VEL
LIN {X 0,Y 544.645,Z 346.932,A -85,B 0,C 180,E1 -3513.698,E2 -3513.698} C_VEL
LIN {X 0,Y 544.599,Z 346.527,A -85,B 0,C 180,E1 -3515.182,E2 -3515.182} C_VEL
LIN {X 0,Y 544.634,Z 344.847,A -85,B 0,C 180,E1 -3516.476,E2 -3516.476} C_VEL
LIN {X 0,Y 544.648,Z 341.839,A -85,B 0,C 180,E1 -3517.786,E2 -3517.786} C_VEL
LIN {X 0,Y 544.675,Z 338.181,A -85,B 0,C 180,E1 -3518.906,E2 -3518.906} C_VEL
LIN {X 0,Y 544.734,Z 333.387,A -85,B 0,C 180,E1 -3520.029,E2 -3520.029} C_VEL
LIN {X 0,Y 544.845,Z 327.309,A -85,B 0,C 180,E1 -3521.155,E2 -3521.155} C_VEL
LIN {X 0,Y 544.959,Z 319.723,A -85,B 0,C 180,E1 -3522.285,E2 -3522.285} C_VEL
LIN {X 0,Y 545.116,Z 311.952,A -85,B 0,C 180,E1 -3523.228,E2 -3523.228} C_VEL
LIN {X 0,Y 545.311,Z 302.438,A -85,B 0,C 180,E1 -3524.173,E2 -3524.173} C_VEL
LIN {X 0,Y 545.488,Z 291.895,A -85,B 0,C 180,E1 -3525.027,E2 -3525.027} C_VEL
LIN {X 0,Y 545.704,Z 280.114,A -85,B 0,C 180,E1 -3525.786,E2 -3525.786} C_VEL
LIN {X 0,Y 545.872,Z 268.574,A -85,B 0,C 180,E1 -3526.357,E2 -3526.357} C_VEL
LIN {X 0,Y 546.126,Z 255.487,A -85,B 0,C 180,E1 -3526.83,E2 -3526.83} C_VEL
LIN {X 0,Y 545.646,Z 249.672,A -85,B 0,C 180,E1 -3527.002,E2 -3527.002} C_VEL
LIN {X 0,Y 544.629,Z 244.001,A -85,B 0,C 180,E1 -3527.167,E2 -3527.167} C_VEL
LIN {X 0,Y 544.61,Z 240.35,A -85,B 0,C 180,E1 -3530.39,E2 -3530.39} C_VEL
LIN {X 0,Y 544.626,Z 237.636,A -85,B 0,C 180,E1 -3532.775,E2 -3532.775} C_VEL
LIN {X 0,Y 544.716,Z 234.558,A -85,B 0,C 180,E1 -3535.424,E2 -3535.424} C_VEL
LIN {X 0,Y 544.733,Z 232.018,A -85,B 0,C 180,E1 -3537.674,E2 -3537.674} C_VEL
LIN {X 0,Y 544.793,Z 229.175,A -85,B 0,C 180,E1 -3540.205,E2 -3540.205} C_VEL
LIN {X 0,Y 544.783,Z 226.07,A -85,B 0,C 180,E1 -3543.014,E2 -3543.014} C_VEL
LIN {X 0,Y 544.82,Z 223.193,A -85,B 0,C 180,E1 -3545.641,E2 -3545.641} C_VEL
LIN {X 0,Y 544.875,Z 220.617,A -85,B 0,C 180,E1 -3548.112,E2 -3548.112} C_VEL
LIN {X 0,Y 545.073,Z 220.586,A -85,B 0,C 180,E1 -3550.471,E2 -3550.471} C_VEL
LIN {X 0,Y 545.073,Z 220.588,A -85,B 0,C 180,E1 -3553.105,E2 -3553.105} C_VEL
LIN {X 0,Y 545.043,Z 220.594,A -85,B 0,C 180,E1 -3556.225,E2 -3556.225} C_VEL
LIN {X 0,Y 545.065,Z 220.589,A -85,B 0,C 180,E1 -3558.883,E2 -3558.883} C_VEL
LIN {X 0,Y 545.074,Z 220.591,A -85,B 0,C 180,E1 -3560.817,E2 -3560.817} C_VEL
LIN {X 0,Y 545.048,Z 220.589,A -85,B 0,C 180,E1 -3563.62,E2 -3563.62} C_VEL
LIN {X 0,Y 545.044,Z 220.591,A -85,B 0,C 180,E1 -3566.326,E2 -3566.326} C_VEL
LIN {X 0,Y 545.054,Z 220.592,A -85,B 0,C 180,E1 -3568.951,E2 -3568.951} C_VEL
LIN {X 0,Y 545.094,Z 220.583,A -85,B 0,C 180,E1 -3571.507,E2 -3571.507} C_VEL
LIN {X 0,Y 545.091,Z 220.586,A -85,B 0,C 180,E1 -3574.489,E2 -3574.489} C_VEL
LIN {X 0,Y 545.033,Z 220.595,A -85,B 0,C 180,E1 -3577.242,E2 -3577.242} C_VEL
LIN {X 0,Y 545.105,Z 220.585,A -85,B 0,C 180,E1 -3580.414,E2 -3580.414} C_VEL
LIN {X 0,Y 545.065,Z 220.588,A -85,B 0,C 180,E1 -3583.521,E2 -3583.521} C_VEL
LIN {X 0,Y 545.085,Z 220.589,A -85,B 0,C 180,E1 -3585.82,E2 -3585.82} C_VEL
LIN {X 0,Y 545.109,Z 220.587,A -85,B 0,C 180,E1 -3588.849,E2 -3588.849} C_VEL
LIN {X 0,Y 545.116,Z 220.582,A -85,B 0,C 180,E1 -3591.847,E2 -3591.847} C_VEL
LIN {X 0,Y 545.205,Z 220.57,A -85,B 0,C 180,E1 -3594.823,E2 -3594.823} C_VEL
LIN {X 0,Y 545.179,Z 220.573,A -85,B 0,C 180,E1 -3597.784,E2 -3597.784} C_VEL
LIN {X 0,Y 545.199,Z 220.574,A -85,B 0,C 180,E1 -3600.739,E2 -3600.739} C_VEL
LIN {X 0,Y 545.162,Z 220.575,A -85,B 0,C 180,E1 -3602.956,E2 -3602.956} C_VEL
LIN {X 0,Y 545.164,Z 220.576,A -85,B 0,C 180,E1 -3605.92,E2 -3605.92} C_VEL
LIN {X 0,Y 545.107,Z 220.586,A -85,B 0,C 180,E1 -3608.9,E2 -3608.9} C_VEL
LIN {X 0,Y 545.122,Z 220.585,A -85,B 0,C 180,E1 -3611.904,E2 -3611.904} C_VEL
LIN {X 0,Y 545.075,Z 220.588,A -85,B 0,C 180,E1 -3614.944,E2 -3614.944} C_VEL
LIN {X 0,Y 545.074,Z 220.586,A -85,B 0,C 180,E1 -3618.026,E2 -3618.026} C_VEL
LIN {X 0,Y 545.083,Z 220.59,A -85,B 0,C 180,E1 -3620.373,E2 -3620.373} C_VEL
LIN {X 0,Y 545.066,Z 220.594,A -85,B 0,C 180,E1 -3623.56,E2 -3623.56} C_VEL
LIN {X 0,Y 545.08,Z 220.585,A -85,B 0,C 180,E1 -3626.001,E2 -3626.001} C_VEL
LIN {X 0,Y 545.084,Z 220.588,A -85,B 0,C 180,E1 -3628.75,E2 -3628.75} C_VEL
LIN {X 0,Y 545.058,Z 220.588,A -85,B 0,C 180,E1 -3631.048,E2 -3631.048} C_VEL
LIN {X 0,Y 545.055,Z 220.592,A -85,B 0,C 180,E1 -3633.673,E2 -3633.673} C_VEL
LIN {X 0,Y 545.061,Z 220.591,A -85,B 0,C 180,E1 -3636.927,E2 -3636.927} C_VEL
LIN {X 0,Y 545.066,Z 220.592,A -85,B 0,C 180,E1 -3640.143,E2 -3640.143} C_VEL
LIN {X 0,Y 545.038,Z 220.591,A -85,B 0,C 180,E1 -3642.696,E2 -3642.696} C_VEL
LIN {X 0,Y 545.052,Z 220.594,A -85,B 0,C 180,E1 -3645.168,E2 -3645.168} C_VEL
LIN {X 0,Y 545.077,Z 220.589,A -85,B 0,C 180,E1 -3647.899,E2 -3647.899} C_VEL
LIN {X 0,Y 545.1,Z 220.586,A -85,B 0,C 180,E1 -3650.677,E2 -3650.677} C_VEL
LIN {X 0,Y 545.058,Z 220.652,A -85,B 0,C 180,E1 -3652.292,E2 -3652.292} C_VEL
LIN {X 0,Y 545.904,Z 225.912,A -85,B 0,C 180,E1 -3654.2,E2 -3654.2} C_VEL
LIN {X 0,Y 545.932,Z 232.486,A -85,B 0,C 180,E1 -3656.39,E2 -3656.39} C_VEL
LIN {X 0,Y 545.751,Z 240.456,A -85,B 0,C 180,E1 -3658.997,E2 -3658.997} C_VEL
LIN {X 0,Y 545.56,Z 249.723,A -85,B 0,C 180,E1 -3661.954,E2 -3661.954} C_VEL
LIN {X 0,Y 545.365,Z 258.99,A -85,B 0,C 180,E1 -3664.834,E2 -3664.834} C_VEL
LIN {X 0,Y 545.219,Z 268.258,A -85,B 0,C 180,E1 -3667.651,E2 -3667.651} C_VEL
LIN {X 0,Y 545.078,Z 277.525,A -85,B 0,C 180,E1 -3670.415,E2 -3670.415} C_VEL
LIN {X 0,Y 544.951,Z 286.792,A -85,B 0,C 180,E1 -3673.133,E2 -3673.133} C_VEL
LIN {X 0,Y 544.837,Z 296.059,A -85,B 0,C 180,E1 -3675.814,E2 -3675.814} C_VEL
LIN {X 0,Y 544.802,Z 299.534,A -85,B 0,C 180,E1 -3676.812,E2 -3676.812} C_VEL
LIN {X 0,Y 546.177,Z 309.484,A -85,B 0,C 180,E1 -3677.058,E2 -3677.058} C_VEL
LIN {X 0,Y 546.005,Z 322.507,A -85,B 0,C 180,E1 -3677.456,E2 -3677.456} C_VEL
LIN {X 0,Y 545.792,Z 333.511,A -85,B 0,C 180,E1 -3677.923,E2 -3677.923} C_VEL
LIN {X 0,Y 545.583,Z 344.168,A -85,B 0,C 180,E1 -3678.506,E2 -3678.506} C_VEL
LIN {X 0,Y 545.424,Z 354.762,A -85,B 0,C 180,E1 -3679.233,E2 -3679.233} C_VEL
LIN {X 0,Y 545.224,Z 365.614,A -85,B 0,C 180,E1 -3680.167,E2 -3680.167} C_VEL
LIN {X 0,Y 545.05,Z 374.423,A -85,B 0,C 180,E1 -3681.1,E2 -3681.1} C_VEL
LIN {X 0,Y 544.894,Z 383.008,A -85,B 0,C 180,E1 -3682.218,E2 -3682.218} C_VEL
LIN {X 0,Y 544.744,Z 390.356,A -85,B 0,C 180,E1 -3683.422,E2 -3683.422} C_VEL
LIN {X 0,Y 544.741,Z 395.371,A -85,B 0,C 180,E1 -3684.448,E2 -3684.448} C_VEL
LIN {X 0,Y 544.66,Z 399.681,A -85,B 0,C 180,E1 -3685.561,E2 -3685.561} C_VEL
LIN {X 0,Y 544.669,Z 401.96,A -85,B 0,C 180,E1 -3686.302,E2 -3686.302} C_VEL
LIN {X 0,Y 544.65,Z 403.811,A -85,B 0,C 180,E1 -3687.042,E2 -3687.042} C_VEL
LIN {X 0,Y 544.546,Z 406.187,A -85,B 0,C 180,E1 -3688.522,E2 -3688.522} C_VEL
LIN {X 0,Y 544.541,Z 407,A -85,B 0,C 180,E1 -3690.001,E2 -3690.001} C_VEL
LIN {X 0,Y 544.546,Z 406.185,A -85,B 0,C 180,E1 -3691.48,E2 -3691.48} C_VEL
LIN {X 0,Y 544.651,Z 403.807,A -85,B 0,C 180,E1 -3692.96,E2 -3692.96} C_VEL
LIN {X 0,Y 544.684,Z 400.893,A -85,B 0,C 180,E1 -3694.071,E2 -3694.071} C_VEL
LIN {X 0,Y 544.654,Z 396.945,A -85,B 0,C 180,E1 -3695.183,E2 -3695.183} C_VEL
LIN {X 0,Y 544.737,Z 391.593,A -85,B 0,C 180,E1 -3696.349,E2 -3696.349} C_VEL
LIN {X 0,Y 544.861,Z 384.231,A -85,B 0,C 180,E1 -3697.598,E2 -3697.598} C_VEL
LIN {X 0,Y 545.027,Z 375.982,A -85,B 0,C 180,E1 -3698.716,E2 -3698.716} C_VEL
LIN {X 0,Y 545.165,Z 367.528,A -85,B 0,C 180,E1 -3699.649,E2 -3699.649} C_VEL
LIN {X 0,Y 545.382,Z 357.084,A -85,B 0,C 180,E1 -3700.582,E2 -3700.582} C_VEL
LIN {X 0,Y 545.589,Z 345.649,A -85,B 0,C 180,E1 -3701.402,E2 -3701.402} C_VEL
LIN {X 0,Y 545.756,Z 335.391,A -85,B 0,C 180,E1 -3701.986,E2 -3701.986} C_VEL
LIN {X 0,Y 545.948,Z 323.735,A -85,B 0,C 180,E1 -3702.5,E2 -3702.5} C_VEL
LIN {X 0,Y 546.136,Z 310.309,A -85,B 0,C 180,E1 -3702.921,E2 -3702.921} C_VEL
LIN {X 0,Y 545.897,Z 306.319,A -85,B 0,C 180,E1 -3703.021,E2 -3703.021} C_VEL
LIN {X 0,Y 544.799,Z 299.527,A -85,B 0,C 180,E1 -3703.19,E2 -3703.19} C_VEL
LIN {X 0,Y 544.934,Z 289.432,A -85,B 0,C 180,E1 -3706.099,E2 -3706.099} C_VEL
LIN {X 0,Y 545.068,Z 278.841,A -85,B 0,C 180,E1 -3709.196,E2 -3709.196} C_VEL
LIN {X 0,Y 545.22,Z 268.25,A -85,B 0,C 180,E1 -3712.351,E2 -3712.351} C_VEL
LIN {X 0,Y 545.359,Z 258.983,A -85,B 0,C 180,E1 -3715.169,E2 -3715.169} C_VEL
LIN {X 0,Y 545.566,Z 249.715,A -85,B 0,C 180,E1 -3718.048,E2 -3718.048} C_VEL
LIN {X 0,Y 545.742,Z 240.448,A -85,B 0,C 180,E1 -3721.006,E2 -3721.006} C_VEL
LIN {X 0,Y 545.936,Z 232.506,A -85,B 0,C 180,E1 -3723.612,E2 -3723.612} C_VEL
LIN {X 0,Y 545.904,Z 225.868,A -85,B 0,C 180,E1 -3725.8,E2 -3725.8} C_VEL
LIN {X 0,Y 545.048,Z 220.595,A -85,B 0,C 180,E1 -3727.77,E2 -3727.77} C_VEL
LIN {X 0,Y 545.085,Z 220.591,A -85,B 0,C 180,E1 -3730.473,E2 -3730.473} C_VEL
LIN {X 0,Y 545.085,Z 220.585,A -85,B 0,C 180,E1 -3733.107,E2 -3733.107} C_VEL
LIN {X 0,Y 545.074,Z 220.588,A -85,B 0,C 180,E1 -3736.225,E2 -3736.225} C_VEL
LIN {X 0,Y 545.088,Z 220.586,A -85,B 0,C 180,E1 -3738.886,E2 -3738.886} C_VEL
LIN {X 0,Y 545.052,Z 220.588,A -85,B 0,C 180,E1 -3741.865,E2 -3741.865} C_VEL
LIN {X 0,Y 545.029,Z 220.596,A -85,B 0,C 180,E1 -3744.531,E2 -3744.531} C_VEL
LIN {X 0,Y 545.057,Z 220.587,A -85,B 0,C 180,E1 -3747.211,E2 -3747.211} C_VEL
LIN {X 0,Y 545.068,Z 220.591,A -85,B 0,C 180,E1 -3749.811,E2 -3749.811} C_VEL
LIN {X 0,Y 545.066,Z 220.587,A -85,B 0,C 180,E1 -3752.834,E2 -3752.834} C_VEL
LIN {X 0,Y 545.055,Z 220.592,A -85,B 0,C 180,E1 -3755.631,E2 -3755.631} C_VEL
LIN {X 0,Y 545.071,Z 220.592,A -85,B 0,C 180,E1 -3758.837,E2 -3758.837} C_VEL
LIN {X 0,Y 545.055,Z 220.589,A -85,B 0,C 180,E1 -3761.195,E2 -3761.195} C_VEL
LIN {X 0,Y 545.04,Z 220.595,A -85,B 0,C 180,E1 -3764.289,E2 -3764.289} C_VEL
LIN {X 0,Y 545.05,Z 220.588,A -85,B 0,C 180,E1 -3766.58,E2 -3766.58} C_VEL
LIN {X 0,Y 545.074,Z 220.586,A -85,B 0,C 180,E1 -3768.848,E2 -3768.848} C_VEL
LIN {X 0,Y 545.093,Z 220.584,A -85,B 0,C 180,E1 -3771.847,E2 -3771.847} C_VEL
LIN {X 0,Y 545.171,Z 220.574,A -85,B 0,C 180,E1 -3774.081,E2 -3774.081} C_VEL
LIN {X 0,Y 545.176,Z 220.575,A -85,B 0,C 180,E1 -3777.044,E2 -3777.044} C_VEL
LIN {X 0,Y 545.21,Z 220.575,A -85,B 0,C 180,E1 -3780,E2 -3780} C_VEL
LIN {X 0,Y 545.164,Z 220.574,A -85,B 0,C 180,E1 -3782.956,E2 -3782.956} C_VEL
LIN {X 0,Y 545.123,Z 220.58,A -85,B 0,C 180,E1 -3785.92,E2 -3785.92} C_VEL
LIN {X 0,Y 545.094,Z 220.588,A -85,B 0,C 180,E1 -3788.901,E2 -3788.901} C_VEL
LIN {X 0,Y 545.112,Z 220.581,A -85,B 0,C 180,E1 -3791.905,E2 -3791.905} C_VEL
LIN {X 0,Y 545.093,Z 220.584,A -85,B 0,C 180,E1 -3794.944,E2 -3794.944} C_VEL
LIN {X 0,Y 545.078,Z 220.59,A -85,B 0,C 180,E1 -3798.026,E2 -3798.026} C_VEL
LIN {X 0,Y 545.098,Z 220.583,A -85,B 0,C 180,E1 -3800.372,E2 -3800.372} C_VEL
LIN {X 0,Y 545.076,Z 220.588,A -85,B 0,C 180,E1 -3803.56,E2 -3803.56} C_VEL
LIN {X 0,Y 545.042,Z 220.595,A -85,B 0,C 180,E1 -3806.828,E2 -3806.828} C_VEL
LIN {X 0,Y 545.033,Z 220.59,A -85,B 0,C 180,E1 -3809.341,E2 -3809.341} C_VEL
LIN {X 0,Y 545.062,Z 220.592,A -85,B 0,C 180,E1 -3811.915,E2 -3811.915} C_VEL
LIN {X 0,Y 545.066,Z 220.587,A -85,B 0,C 180,E1 -3814.565,E2 -3814.565} C_VEL
LIN {X 0,Y 545.069,Z 220.588,A -85,B 0,C 180,E1 -3816.955,E2 -3816.955} C_VEL
LIN {X 0,Y 544.361,Z 220.68,A -85,B 0,C 180,E1 -3817.572,E2 -3817.572} C_VEL
LIN {X 0,Y 541.501,Z 221.034,A -85,B 0,C 180,E1 -3818.573,E2 -3818.573} C_VEL
LIN {X 0,Y 539.112,Z 221.333,A -85,B 0,C 180,E1 -3819.378,E2 -3819.378} C_VEL
LIN {X 0,Y 538.093,Z 221.456,A -85,B 0,C 180,E1 -3820,E2 -3820} C_VEL
LIN {X 0,Y 538.011,Z 221.466,A -85,B 0,C 180,E1 -3820.211,E2 -3820.211} C_VEL
LIN {X 0,Y 537.987,Z 221.472,A -85,B 0,C 180,E1 -3822.982,E2 -3822.982} C_VEL
LIN {X 0,Y 538.002,Z 221.469,A -85,B 0,C 180,E1 -3825.929,E2 -3825.929} C_VEL
LIN {X 0,Y 537.985,Z 221.473,A -85,B 0,C 180,E1 -3828.221,E2 -3828.221} C_VEL
LIN {X 0,Y 538.01,Z 221.467,A -85,B 0,C 180,E1 -3831.168,E2 -3831.168} C_VEL
LIN {X 0,Y 537.997,Z 221.468,A -85,B 0,C 180,E1 -3834.089,E2 -3834.089} C_VEL
LIN {X 0,Y 538.038,Z 221.467,A -85,B 0,C 180,E1 -3836.727,E2 -3836.727} C_VEL
LIN {X 0,Y 537.889,Z 221.487,A -85,B 0,C 180,E1 -3839.582,E2 -3839.582} C_VEL
LIN {X 0,Y 537.8,Z 221.498,A -85,B 0,C 180,E1 -3840.225,E2 -3840.225} C_VEL
LIN {X 0,Y 537.728,Z 224.103,A -85,B 0,C 180,E1 -3842.777,E2 -3842.777} C_VEL
LIN {X 0,Y 537.73,Z 226.871,A -85,B 0,C 180,E1 -3845.276,E2 -3845.276} C_VEL
LIN {X 0,Y 537.661,Z 230.494,A -85,B 0,C 180,E1 -3848.53,E2 -3848.53} C_VEL
LIN {X 0,Y 537.629,Z 233.226,A -85,B 0,C 180,E1 -3850.924,E2 -3850.924} C_VEL
LIN {X 0,Y 537.621,Z 235.848,A -85,B 0,C 180,E1 -3853.285,E2 -3853.285} C_VEL
LIN {X 0,Y 537.604,Z 238.486,A -85,B 0,C 180,E1 -3855.617,E2 -3855.617} C_VEL
LIN {X 0,Y 537.65,Z 242.031,A -85,B 0,C 180,E1 -3858.691,E2 -3858.691} C_VEL
LIN {X 0,Y 537.539,Z 244.433,A -85,B 0,C 180,E1 -3860.759,E2 -3860.759} C_VEL
LIN {X 0,Y 539.239,Z 254.434,A -85,B 0,C 180,E1 -3861.048,E2 -3861.048} C_VEL
LIN {X 0,Y 539.016,Z 267.634,A -85,B 0,C 180,E1 -3861.517,E2 -3861.517} C_VEL
LIN {X 0,Y 538.826,Z 280.094,A -85,B 0,C 180,E1 -3862.127,E2 -3862.127} C_VEL
LIN {X 0,Y 538.536,Z 291.147,A -85,B 0,C 180,E1 -3862.833,E2 -3862.833} C_VEL
LIN {X 0,Y 538.392,Z 301.101,A -85,B 0,C 180,E1 -3863.628,E2 -3863.628} C_VEL
LIN {X 0,Y 538.13,Z 310.684,A -85,B 0,C 180,E1 -3864.566,E2 -3864.566} C_VEL
LIN {X 0,Y 537.992,Z 318.536,A -85,B 0,C 180,E1 -3865.503,E2 -3865.503} C_VEL
LIN {X 0,Y 537.825,Z 326.255,A -85,B 0,C 180,E1 -3866.628,E2 -3866.628} C_VEL
LIN {X 0,Y 537.568,Z 332.438,A -85,B 0,C 180,E1 -3867.751,E2 -3867.751} C_VEL
LIN {X 0,Y 537.607,Z 337.343,A -85,B 0,C 180,E1 -3868.875,E2 -3868.875} C_VEL
LIN {X 0,Y 537.484,Z 341.164,A -85,B 0,C 180,E1 -3869.999,E2 -3869.999} C_VEL
LIN {X 0,Y 537.453,Z 344.689,A -85,B 0,C 180,E1 -3871.498,E2 -3871.498} C_VEL
LIN {X 0,Y 537.489,Z 345.86,A -85,B 0,C 180,E1 -3872.247,E2 -3872.247} C_VEL
LIN {X 0,Y 537.545,Z 346.594,A -85,B 0,C 180,E1 -3872.997,E2 -3872.997} C_VEL
LIN {X 0,Y 537.561,Z 346.943,A -85,B 0,C 180,E1 -3873.747,E2 -3873.747} C_VEL
LIN {X 0,Y 537.52,Z 346.487,A -85,B 0,C 180,E1 -3875.25,E2 -3875.25} C_VEL
LIN {X 0,Y 537.536,Z 344.948,A -85,B 0,C 180,E1 -3876.452,E2 -3876.452} C_VEL
LIN {X 0,Y 537.556,Z 341.721,A -85,B 0,C 180,E1 -3877.889,E2 -3877.889} C_VEL
LIN {X 0,Y 537.576,Z 338.058,A -85,B 0,C 180,E1 -3879.025,E2 -3879.025} C_VEL
LIN {X 0,Y 537.649,Z 333.265,A -85,B 0,C 180,E1 -3880.163,E2 -3880.163} C_VEL
LIN {X 0,Y 537.813,Z 326.311,A -85,B 0,C 180,E1 -3881.453,E2 -3881.453} C_VEL
LIN {X 0,Y 537.981,Z 318.14,A -85,B 0,C 180,E1 -3882.638,E2 -3882.638} C_VEL
LIN {X 0,Y 538.135,Z 310.03,A -85,B 0,C 180,E1 -3883.595,E2 -3883.595} C_VEL
LIN {X 0,Y 538.346,Z 300.588,A -85,B 0,C 180,E1 -3884.509,E2 -3884.509} C_VEL
LIN {X 0,Y 538.547,Z 290.27,A -85,B 0,C 180,E1 -3885.322,E2 -3885.322} C_VEL
LIN {X 0,Y 538.791,Z 279.544,A -85,B 0,C 180,E1 -3885.994,E2 -3885.994} C_VEL
LIN {X 0,Y 539.008,Z 266.563,A -85,B 0,C 180,E1 -3886.62,E2 -3886.62} C_VEL
LIN {X 0,Y 539.198,Z 253.536,A -85,B 0,C 180,E1 -3887.068,E2 -3887.068} C_VEL
LIN {X 0,Y 537.54,Z 244.387,A -85,B 0,C 180,E1 -3887.331,E2 -3887.331} C_VEL
LIN {X 0,Y 537.545,Z 241.539,A -85,B 0,C 180,E1 -3889.871,E2 -3889.871} C_VEL
LIN {X 0,Y 537.548,Z 238.795,A -85,B 0,C 180,E1 -3892.28,E2 -3892.28} C_VEL
LIN {X 0,Y 537.606,Z 235.97,A -85,B 0,C 180,E1 -3894.728,E2 -3894.728} C_VEL
LIN {X 0,Y 537.659,Z 233.091,A -85,B 0,C 180,E1 -3897.269,E2 -3897.269} C_VEL
LIN {X 0,Y 537.708,Z 229.626,A -85,B 0,C 180,E1 -3900.385,E2 -3900.385} C_VEL
LIN {X 0,Y 537.724,Z 226.453,A -85,B 0,C 180,E1 -3903.292,E2 -3903.292} C_VEL
LIN {X 0,Y 537.768,Z 223.481,A -85,B 0,C 180,E1 -3906.02,E2 -3906.02} C_VEL
LIN {X 0,Y 537.805,Z 221.498,A -85,B 0,C 180,E1 -3907.892,E2 -3907.892} C_VEL
LIN {X 0,Y 538.044,Z 221.464,A -85,B 0,C 180,E1 -3910.774,E2 -3910.774} C_VEL
LIN {X 0,Y 538.024,Z 221.467,A -85,B 0,C 180,E1 -3914.073,E2 -3914.073} C_VEL
LIN {X 0,Y 537.991,Z 221.469,A -85,B 0,C 180,E1 -3917.015,E2 -3917.015} C_VEL
LIN {X 0,Y 538.039,Z 221.468,A -85,B 0,C 180,E1 -3919.252,E2 -3919.252} C_VEL
LIN {X 0,Y 537.986,Z 221.47,A -85,B 0,C 180,E1 -3922.121,E2 -3922.121} C_VEL
LIN {X 0,Y 538.011,Z 221.466,A -85,B 0,C 180,E1 -3924.916,E2 -3924.916} C_VEL
LIN {X 0,Y 538.007,Z 221.472,A -85,B 0,C 180,E1 -3927.616,E2 -3927.616} C_VEL
LIN {X 0,Y 538.005,Z 221.467,A -85,B 0,C 180,E1 -3930.238,E2 -3930.238} C_VEL
LIN {X 0,Y 538.063,Z 221.461,A -85,B 0,C 180,E1 -3932.796,E2 -3932.796} C_VEL
LIN {X 0,Y 538.04,Z 221.463,A -85,B 0,C 180,E1 -3935.292,E2 -3935.292} C_VEL
LIN {X 0,Y 538.005,Z 221.467,A -85,B 0,C 180,E1 -3938.041,E2 -3938.041} C_VEL
LIN {X 0,Y 538.021,Z 221.468,A -85,B 0,C 180,E1 -3940.939,E2 -3940.939} C_VEL
LIN {X 0,Y 538.015,Z 221.465,A -85,B 0,C 180,E1 -3943.299,E2 -3943.299} C_VEL
LIN {X 0,Y 538.054,Z 221.467,A -85,B 0,C 180,E1 -3945.63,E2 -3945.63} C_VEL
LIN {X 0,Y 538.068,Z 221.462,A -85,B 0,C 180,E1 -3948.701,E2 -3948.701} C_VEL
LIN {X 0,Y 538.072,Z 221.459,A -85,B 0,C 180,E1 -3951.739,E2 -3951.739} C_VEL
LIN {X 0,Y 538.181,Z 221.445,A -85,B 0,C 180,E1 -3954.755,E2 -3954.755} C_VEL
LIN {X 0,Y 538.152,Z 221.449,A -85,B 0,C 180,E1 -3957.755,E2 -3957.755} C_VEL
LIN {X 0,Y 538.169,Z 221.449,A -85,B 0,C 180,E1 -3960.748,E2 -3960.748} C_VEL
LIN {X 0,Y 538.128,Z 221.451,A -85,B 0,C 180,E1 -3962.994,E2 -3962.994} C_VEL
LIN {X 0,Y 538.116,Z 221.453,A -85,B 0,C 180,E1 -3965.997,E2 -3965.997} C_VEL
LIN {X 0,Y 538.057,Z 221.463,A -85,B 0,C 180,E1 -3969.018,E2 -3969.018} C_VEL
LIN {X 0,Y 538.07,Z 221.464,A -85,B 0,C 180,E1 -3972.063,E2 -3972.063} C_VEL
LIN {X 0,Y 538.035,Z 221.467,A -85,B 0,C 180,E1 -3975.144,E2 -3975.144} C_VEL
LIN {X 0,Y 538.026,Z 221.466,A -85,B 0,C 180,E1 -3978.27,E2 -3978.27} C_VEL
LIN {X 0,Y 538.027,Z 221.466,A -85,B 0,C 180,E1 -3980.652,E2 -3980.652} C_VEL
LIN {X 0,Y 537.99,Z 221.471,A -85,B 0,C 180,E1 -3983.889,E2 -3983.889} C_VEL
LIN {X 0,Y 538.041,Z 221.463,A -85,B 0,C 180,E1 -3986.367,E2 -3986.367} C_VEL
LIN {X 0,Y 538.047,Z 221.463,A -85,B 0,C 180,E1 -3988.939,E2 -3988.939} C_VEL
LIN {X 0,Y 537.999,Z 221.473,A -85,B 0,C 180,E1 -3991.888,E2 -3991.888} C_VEL
LIN {X 0,Y 538.002,Z 221.469,A -85,B 0,C 180,E1 -3994.619,E2 -3994.619} C_VEL
LIN {X 0,Y 537.996,Z 221.469,A -85,B 0,C 180,E1 -3997.171,E2 -3997.171} C_VEL
LIN {X 0,Y 538.022,Z 221.468,A -85,B 0,C 180,E1 -3999.797,E2 -3999.797} C_VEL
LIN {X 0,Y 537.99,Z 221.47,A -85,B 0,C 180,E1 -4002.789,E2 -4002.789} C_VEL
LIN {X 0,Y 538.022,Z 221.47,A -85,B 0,C 180,E1 -4005.141,E2 -4005.141} C_VEL
LIN {X 0,Y 538.035,Z 221.469,A -85,B 0,C 180,E1 -4008.229,E2 -4008.229} C_VEL
LIN {X 0,Y 538.054,Z 221.465,A -85,B 0,C 180,E1 -4010.413,E2 -4010.413} C_VEL
LIN {X 0,Y 538.029,Z 221.572,A -85,B 0,C 180,E1 -4012.063,E2 -4012.063} C_VEL
LIN {X 0,Y 538.912,Z 226.967,A -85,B 0,C 180,E1 -4014.068,E2 -4014.068} C_VEL
LIN {X 0,Y 538.957,Z 233.504,A -85,B 0,C 180,E1 -4016.278,E2 -4016.278} C_VEL
LIN {X 0,Y 538.766,Z 241.78,A -85,B 0,C 180,E1 -4018.987,E2 -4018.987} C_VEL
LIN {X 0,Y 538.578,Z 251.047,A -85,B 0,C 180,E1 -4021.982,E2 -4021.982} C_VEL
LIN {X 0,Y 538.343,Z 260.314,A -85,B 0,C 180,E1 -4024.896,E2 -4024.896} C_VEL
LIN {X 0,Y 538.2,Z 269.581,A -85,B 0,C 180,E1 -4027.749,E2 -4027.749} C_VEL
LIN {X 0,Y 538.02,Z 278.849,A -85,B 0,C 180,E1 -4030.544,E2 -4030.544} C_VEL
LIN {X 0,Y 537.89,Z 288.116,A -85,B 0,C 180,E1 -4033.296,E2 -4033.296} C_VEL
LIN {X 0,Y 537.776,Z 297.383,A -85,B 0,C 180,E1 -4036.01,E2 -4036.01} C_VEL
LIN {X 0,Y 537.744,Z 299.576,A -85,B 0,C 180,E1 -4036.648,E2 -4036.648} C_VEL
LIN {X 0,Y 539.249,Z 309.484,A -85,B 0,C 180,E1 -4036.889,E2 -4036.889} C_VEL
LIN {X 0,Y 539.09,Z 322.507,A -85,B 0,C 180,E1 -4037.292,E2 -4037.292} C_VEL
LIN {X 0,Y 538.852,Z 333.512,A -85,B 0,C 180,E1 -4037.765,E2 -4037.765} C_VEL
LIN {X 0,Y 538.595,Z 344.866,A -85,B 0,C 180,E1 -4038.397,E2 -4038.397} C_VEL
LIN {X 0,Y 538.41,Z 355.94,A -85,B 0,C 180,E1 -4039.186,E2 -4039.186} C_VEL
LIN {X 0,Y 538.221,Z 365.614,A -85,B 0,C 180,E1 -4040.038,E2 -4040.038} C_VEL
LIN {X 0,Y 538.014,Z 374.423,A -85,B 0,C 180,E1 -4040.983,E2 -4040.983} C_VEL
LIN {X 0,Y 537.828,Z 383.009,A -85,B 0,C 180,E1 -4042.115,E2 -4042.115} C_VEL
LIN {X 0,Y 537.704,Z 389.874,A -85,B 0,C 180,E1 -4043.246,E2 -4043.246} C_VEL
LIN {X 0,Y 537.676,Z 395.371,A -85,B 0,C 180,E1 -4044.375,E2 -4044.375} C_VEL
LIN {X 0,Y 537.557,Z 399.681,A -85,B 0,C 180,E1 -4045.502,E2 -4045.502} C_VEL
LIN {X 0,Y 537.591,Z 401.96,A -85,B 0,C 180,E1 -4046.253,E2 -4046.253} C_VEL
LIN {X 0,Y 537.551,Z 403.811,A -85,B 0,C 180,E1 -4047.003,E2 -4047.003} C_VEL
LIN {X 0,Y 537.49,Z 405.2,A -85,B 0,C 180,E1 -4047.753,E2 -4047.753} C_VEL
LIN {X 0,Y 537.442,Z 406.786,A -85,B 0,C 180,E1 -4049.252,E2 -4049.252} C_VEL
LIN {X 0,Y 537.442,Z 407,A -85,B 0,C 180,E1 -4050.001,E2 -4050.001} C_VEL
LIN {X 0,Y 537.451,Z 406.185,A -85,B 0,C 180,E1 -4051.5,E2 -4051.5} C_VEL
LIN {X 0,Y 537.49,Z 405.198,A -85,B 0,C 180,E1 -4052.249,E2 -4052.249} C_VEL
LIN {X 0,Y 537.551,Z 403.807,A -85,B 0,C 180,E1 -4052.999,E2 -4052.999} C_VEL
LIN {X 0,Y 537.604,Z 400.893,A -85,B 0,C 180,E1 -4054.124,E2 -4054.124} C_VEL
LIN {X 0,Y 537.588,Z 396.945,A -85,B 0,C 180,E1 -4055.252,E2 -4055.252} C_VEL
LIN {X 0,Y 537.652,Z 392.085,A -85,B 0,C 180,E1 -4056.334,E2 -4056.334} C_VEL
LIN {X 0,Y 537.792,Z 385.462,A -85,B 0,C 180,E1 -4057.51,E2 -4057.51} C_VEL
LIN {X 0,Y 537.97,Z 377.47,A -85,B 0,C 180,E1 -4058.642,E2 -4058.642} C_VEL
LIN {X 0,Y 538.119,Z 369.326,A -85,B 0,C 180,E1 -4059.587,E2 -4059.587} C_VEL
LIN {X 0,Y 538.338,Z 359.389,A -85,B 0,C 180,E1 -4060.532,E2 -4060.532} C_VEL
LIN {X 0,Y 538.533,Z 349.571,A -85,B 0,C 180,E1 -4061.29,E2 -4061.29} C_VEL
LIN {X 0,Y 538.742,Z 338.57,A -85,B 0,C 180,E1 -4061.972,E2 -4061.972} C_VEL
LIN {X 0,Y 538.98,Z 326.085,A -85,B 0,C 180,E1 -4062.569,E2 -4062.569} C_VEL
LIN {X 0,Y 539.202,Z 313.051,A -85,B 0,C 180,E1 -4063.018,E2 -4063.018} C_VEL
LIN {X 0,Y 539.022,Z 307.458,A -85,B 0,C 180,E1 -4063.167,E2 -4063.167} C_VEL
LIN {X 0,Y 537.731,Z 299.527,A -85,B 0,C 180,E1 -4063.367,E2 -4063.367} C_VEL
LIN {X 0,Y 537.875,Z 289.432,A -85,B 0,C 180,E1 -4066.316,E2 -4066.316} C_VEL
LIN {X 0,Y 537.995,Z 280.165,A -85,B 0,C 180,E1 -4069.063,E2 -4069.063} C_VEL
LIN {X 0,Y 538.131,Z 272.221,A -85,B 0,C 180,E1 -4071.45,E2 -4071.45} C_VEL
LIN {X 0,Y 538.331,Z 262.956,A -85,B 0,C 180,E1 -4074.283,E2 -4074.283} C_VEL
LIN {X 0,Y 538.527,Z 252.843,A -85,B 0,C 180,E1 -4077.448,E2 -4077.448} C_VEL
LIN {X 0,Y 538.729,Z 243.096,A -85,B 0,C 180,E1 -4080.583,E2 -4080.583} C_VEL
LIN {X 0,Y 538.915,Z 235.109,A -85,B 0,C 180,E1 -4083.212,E2 -4083.212} C_VEL
LIN {X 0,Y 538.988,Z 228.276,A -85,B 0,C 180,E1 -4085.469,E2 -4085.469} C_VEL
LIN {X 0,Y 538.387,Z 223.479,A -85,B 0,C 180,E1 -4087.223,E2 -4087.223} C_VEL
LIN {X 0,Y 537.999,Z 221.473,A -85,B 0,C 180,E1 -4088.006,E2 -4088.006} C_VEL
LIN {X 0,Y 538.028,Z 221.469,A -85,B 0,C 180,E1 -4090.779,E2 -4090.779} C_VEL
LIN {X 0,Y 538.011,Z 221.472,A -85,B 0,C 180,E1 -4093.816,E2 -4093.816} C_VEL
LIN {X 0,Y 538.028,Z 221.466,A -85,B 0,C 180,E1 -4096.186,E2 -4096.186} C_VEL
LIN {X 0,Y 538.055,Z 221.466,A -85,B 0,C 180,E1 -4099.253,E2 -4099.253} C_VEL
LIN {X 0,Y 537.994,Z 221.467,A -85,B 0,C 180,E1 -4102.122,E2 -4102.122} C_VEL
LIN {X 0,Y 537.991,Z 221.471,A -85,B 0,C 180,E1 -4104.915,E2 -4104.915} C_VEL
LIN {X 0,Y 538.011,Z 221.465,A -85,B 0,C 180,E1 -4107.617,E2 -4107.617} C_VEL
LIN {X 0,Y 538.012,Z 221.47,A -85,B 0,C 180,E1 -4110.238,E2 -4110.238} C_VEL
LIN {X 0,Y 538.037,Z 221.463,A -85,B 0,C 180,E1 -4112.795,E2 -4112.795} C_VEL
LIN {X 0,Y 538.029,Z 221.468,A -85,B 0,C 180,E1 -4115.292,E2 -4115.292} C_VEL
LIN {X 0,Y 538.022,Z 221.464,A -85,B 0,C 180,E1 -4118.042,E2 -4118.042} C_VEL
LIN {X 0,Y 538.088,Z 221.458,A -85,B 0,C 180,E1 -4120.148,E2 -4120.148} C_VEL
LIN {X 0,Y 537.974,Z 221.47,A -85,B 0,C 180,E1 -4123.297,E2 -4123.297} C_VEL
LIN {X 0,Y 538.043,Z 221.464,A -85,B 0,C 180,E1 -4125.63,E2 -4125.63} C_VEL
LIN {X 0,Y 538.027,Z 221.463,A -85,B 0,C 180,E1 -4128.7,E2 -4128.7} C_VEL
LIN {X 0,Y 538.059,Z 221.462,A -85,B 0,C 180,E1 -4131.739,E2 -4131.739} C_VEL
LIN {X 0,Y 538.123,Z 221.452,A -85,B 0,C 180,E1 -4134.003,E2 -4134.003} C_VEL
LIN {X 0,Y 538.143,Z 221.452,A -85,B 0,C 180,E1 -4137.006,E2 -4137.006} C_VEL
LIN {X 0,Y 538.18,Z 221.45,A -85,B 0,C 180,E1 -4140,E2 -4140} C_VEL
LIN {X 0,Y 538.132,Z 221.45,A -85,B 0,C 180,E1 -4142.995,E2 -4142.995} C_VEL
LIN {X 0,Y 538.077,Z 221.457,A -85,B 0,C 180,E1 -4145.998,E2 -4145.998} C_VEL
LIN {X 0,Y 538.048,Z 221.467,A -85,B 0,C 180,E1 -4149.018,E2 -4149.018} C_VEL
LIN {X 0,Y 538.072,Z 221.459,A -85,B 0,C 180,E1 -4152.063,E2 -4152.063} C_VEL
LIN {X 0,Y 538.053,Z 221.461,A -85,B 0,C 180,E1 -4155.144,E2 -4155.144} C_VEL
LIN {X 0,Y 538.032,Z 221.466,A -85,B 0,C 180,E1 -4158.27,E2 -4158.27} C_VEL
LIN {X 0,Y 538.044,Z 221.462,A -85,B 0,C 180,E1 -4160.651,E2 -4160.651} C_VEL
LIN {X 0,Y 538.013,Z 221.465,A -85,B 0,C 180,E1 -4163.877,E2 -4163.877} C_VEL
LIN {X 0,Y 537.974,Z 221.472,A -85,B 0,C 180,E1 -4166.37,E2 -4166.37} C_VEL
LIN {X 0,Y 537.999,Z 221.469,A -85,B 0,C 180,E1 -4168.926,E2 -4168.926} C_VEL
LIN {X 0,Y 538.017,Z 221.469,A -85,B 0,C 180,E1 -4171.887,E2 -4171.887} C_VEL
LIN {X 0,Y 538.016,Z 221.465,A -85,B 0,C 180,E1 -4174.617,E2 -4174.617} C_VEL
LIN {X 0,Y 538.007,Z 221.471,A -85,B 0,C 180,E1 -4177.169,E2 -4177.169} C_VEL
LIN {X 0,Y 538.011,Z 221.466,A -85,B 0,C 180,E1 -4180.211,E2 -4180.211} C_VEL
LIN {X 0,Y 537.348,Z 221.554,A -85,B 0,C 180,E1 -4180.836,E2 -4180.836} C_VEL
LIN {X 0,Y 534.494,Z 221.907,A -85,B 0,C 180,E1 -4181.851,E2 -4181.851} C_VEL
LIN {X 0,Y 532.075,Z 222.211,A -85,B 0,C 180,E1 -4182.668,E2 -4182.668} C_VEL
LIN {X 0,Y 531.031,Z 222.336,A -85,B 0,C 180,E1 -4183.299,E2 -4183.299} C_VEL
LIN {X 0,Y 530.944,Z 222.346,A -85,B 0,C 180,E1 -4183.513,E2 -4183.513} C_VEL
LIN {X 0,Y 530.926,Z 222.351,A -85,B 0,C 180,E1 -4186.5,E2 -4186.5} C_VEL
LIN {X 0,Y 530.923,Z 222.351,A -85,B 0,C 180,E1 -4189.561,E2 -4189.561} C_VEL
LIN {X 0,Y 530.972,Z 222.342,A -85,B 0,C 180,E1 -4192.577,E2 -4192.577} C_VEL
LIN {X 0,Y 530.986,Z 222.346,A -85,B 0,C 180,E1 -4195.309,E2 -4195.309} C_VEL
LIN {X 0,Y 530.947,Z 222.347,A -85,B 0,C 180,E1 -4198.029,E2 -4198.029} C_VEL
LIN {X 0,Y 530.687,Z 222.448,A -85,B 0,C 180,E1 -4200.658,E2 -4200.658} C_VEL
LIN {X 0,Y 530.63,Z 225.275,A -85,B 0,C 180,E1 -4203.235,E2 -4203.235} C_VEL
LIN {X 0,Y 530.663,Z 228.372,A -85,B 0,C 180,E1 -4206.04,E2 -4206.04} C_VEL
LIN {X 0,Y 530.57,Z 231.698,A -85,B 0,C 180,E1 -4209.043,E2 -4209.043} C_VEL
LIN {X 0,Y 530.523,Z 234.43,A -85,B 0,C 180,E1 -4211.461,E2 -4211.461} C_VEL
LIN {X 0,Y 530.54,Z 237.094,A -85,B 0,C 180,E1 -4213.847,E2 -4213.847} C_VEL
LIN {X 0,Y 530.52,Z 239.777,A -85,B 0,C 180,E1 -4216.204,E2 -4216.204} C_VEL
LIN {X 0,Y 530.565,Z 242.517,A -85,B 0,C 180,E1 -4218.588,E2 -4218.588} C_VEL
LIN {X 0,Y 530.492,Z 244.848,A -85,B 0,C 180,E1 -4220.563,E2 -4220.563} C_VEL
LIN {X 0,Y 532.329,Z 255.071,A -85,B 0,C 180,E1 -4220.883,E2 -4220.883} C_VEL
LIN {X 0,Y 532.106,Z 268.207,A -85,B 0,C 180,E1 -4221.358,E2 -4221.358} C_VEL
LIN {X 0,Y 531.937,Z 279.76,A -85,B 0,C 180,E1 -4221.929,E2 -4221.929} C_VEL
LIN {X 0,Y 531.622,Z 290.762,A -85,B 0,C 180,E1 -4222.625,E2 -4222.625} C_VEL
LIN {X 0,Y 531.421,Z 301.073,A -85,B 0,C 180,E1 -4223.449,E2 -4223.449} C_VEL
LIN {X 0,Y 531.133,Z 311.605,A -85,B 0,C 180,E1 -4224.494,E2 -4224.494} C_VEL
LIN {X 0,Y 530.959,Z 319.377,A -85,B 0,C 180,E1 -4225.444,E2 -4225.444} C_VEL
LIN {X 0,Y 530.778,Z 326.994,A -85,B 0,C 180,E1 -4226.583,E2 -4226.583} C_VEL
LIN {X 0,Y 530.507,Z 333.116,A -85,B 0,C 180,E1 -4227.721,E2 -4227.721} C_VEL
LIN {X 0,Y 530.547,Z 337.967,A -85,B 0,C 180,E1 -4228.86,E2 -4228.86} C_VEL
LIN {X 0,Y 530.405,Z 341.739,A -85,B 0,C 180,E1 -4229.999,E2 -4229.999} C_VEL
LIN {X 0,Y 530.37,Z 345.217,A -85,B 0,C 180,E1 -4231.518,E2 -4231.518} C_VEL
LIN {X 0,Y 530.41,Z 346.33,A -85,B 0,C 180,E1 -4232.277,E2 -4232.277} C_VEL
LIN {X 0,Y 530.479,Z 347.023,A -85,B 0,C 180,E1 -4233.037,E2 -4233.037} C_VEL
LIN {X 0,Y 530.479,Z 347.345,A -85,B 0,C 180,E1 -4233.797,E2 -4233.797} C_VEL
LIN {X 0,Y 530.404,Z 347.295,A -85,B 0,C 180,E1 -4234.559,E2 -4234.559} C_VEL
LIN {X 0,Y 530.443,Z 346.839,A -85,B 0,C 180,E1 -4235.32,E2 -4235.32} C_VEL
LIN {X 0,Y 530.468,Z 344.692,A -85,B 0,C 180,E1 -4236.847,E2 -4236.847} C_VEL
LIN {X 0,Y 530.479,Z 341.999,A -85,B 0,C 180,E1 -4237.995,E2 -4237.995} C_VEL
LIN {X 0,Y 530.518,Z 338.285,A -85,B 0,C 180,E1 -4239.146,E2 -4239.146} C_VEL
LIN {X 0,Y 530.611,Z 333.436,A -85,B 0,C 180,E1 -4240.299,E2 -4240.299} C_VEL
LIN {X 0,Y 530.792,Z 326.851,A -85,B 0,C 180,E1 -4241.533,E2 -4241.533} C_VEL
LIN {X 0,Y 530.956,Z 319.633,A -85,B 0,C 180,E1 -4242.614,E2 -4242.614} C_VEL
LIN {X 0,Y 531.115,Z 311.738,A -85,B 0,C 180,E1 -4243.583,E2 -4243.583} C_VEL
LIN {X 0,Y 531.364,Z 302.065,A -85,B 0,C 180,E1 -4244.553,E2 -4244.553} C_VEL
LIN {X 0,Y 531.601,Z 291.272,A -85,B 0,C 180,E1 -4245.429,E2 -4245.429} C_VEL
LIN {X 0,Y 531.865,Z 280.738,A -85,B 0,C 180,E1 -4246.109,E2 -4246.109} C_VEL
LIN {X 0,Y 532.062,Z 267.974,A -85,B 0,C 180,E1 -4246.744,E2 -4246.744} C_VEL
LIN {X 0,Y 532.337,Z 254.813,A -85,B 0,C 180,E1 -4247.215,E2 -4247.215} C_VEL
LIN {X 0,Y 530.472,Z 244.784,A -85,B 0,C 180,E1 -4247.523,E2 -4247.523} C_VEL
LIN {X 0,Y 530.466,Z 241.851,A -85,B 0,C 180,E1 -4250.148,E2 -4250.148} C_VEL
LIN {X 0,Y 530.461,Z 239.022,A -85,B 0,C 180,E1 -4252.594,E2 -4252.594} C_VEL
LIN {X 0,Y 530.54,Z 236.205,A -85,B 0,C 180,E1 -4255.08,E2 -4255.08} C_VEL
LIN {X 0,Y 530.58,Z 233.328,A -85,B 0,C 180,E1 -4257.619,E2 -4257.619} C_VEL
LIN {X 0,Y 530.634,Z 230.076,A -85,B 0,C 180,E1 -4260.582,E2 -4260.582} C_VEL
LIN {X 0,Y 530.675,Z 226.959,A -85,B 0,C 180,E1 -4263.452,E2 -4263.452} C_VEL
LIN {X 0,Y 530.699,Z 224.081,A -85,B 0,C 180,E1 -4266.116,E2 -4266.116} C_VEL
LIN {X 0,Y 530.728,Z 222.576,A -85,B 0,C 180,E1 -4267.526,E2 -4267.526} C_VEL
LIN {X 0,Y 530.931,Z 222.349,A -85,B 0,C 180,E1 -4269.847,E2 -4269.847} C_VEL
LIN {X 0,Y 530.975,Z 222.346,A -85,B 0,C 180,E1 -4272.455,E2 -4272.455} C_VEL
LIN {X 0,Y 530.977,Z 222.344,A -85,B 0,C 180,E1 -4275.62,E2 -4275.62} C_VEL
LIN {X 0,Y 530.979,Z 222.342,A -85,B 0,C 180,E1 -4278.563,E2 -4278.563} C_VEL
LIN {X 0,Y 530.95,Z 222.346,A -85,B 0,C 180,E1 -4281.528,E2 -4281.528} C_VEL
LIN {X 0,Y 530.974,Z 222.347,A -85,B 0,C 180,E1 -4284.381,E2 -4284.381} C_VEL
LIN {X 0,Y 530.957,Z 222.346,A -85,B 0,C 180,E1 -4287.132,E2 -4287.132} C_VEL
LIN {X 0,Y 530.951,Z 222.345,A -85,B 0,C 180,E1 -4289.802,E2 -4289.802} C_VEL
LIN {X 0,Y 531.009,Z 222.343,A -85,B 0,C 180,E1 -4292.465,E2 -4292.465} C_VEL
LIN {X 0,Y 530.999,Z 222.339,A -85,B 0,C 180,E1 -4294.942,E2 -4294.942} C_VEL
LIN {X 0,Y 530.96,Z 222.344,A -85,B 0,C 180,E1 -4298.246,E2 -4298.246} C_VEL
LIN {X 0,Y 530.981,Z 222.348,A -85,B 0,C 180,E1 -4300.677,E2 -4300.677} C_VEL
LIN {X 0,Y 530.976,Z 222.342,A -85,B 0,C 180,E1 -4303.07,E2 -4303.07} C_VEL
LIN {X 0,Y 531.009,Z 222.342,A -85,B 0,C 180,E1 -4305.435,E2 -4305.435} C_VEL
LIN {X 0,Y 531.027,Z 222.337,A -85,B 0,C 180,E1 -4308.549,E2 -4308.549} C_VEL
LIN {X 0,Y 531.041,Z 222.334,A -85,B 0,C 180,E1 -4311.629,E2 -4311.629} C_VEL
LIN {X 0,Y 531.137,Z 222.322,A -85,B 0,C 180,E1 -4314.685,E2 -4314.685} C_VEL
LIN {X 0,Y 531.125,Z 222.324,A -85,B 0,C 180,E1 -4317.725,E2 -4317.725} C_VEL
LIN {X 0,Y 531.139,Z 222.325,A -85,B 0,C 180,E1 -4320.758,E2 -4320.758} C_VEL
LIN {X 0,Y 531.095,Z 222.327,A -85,B 0,C 180,E1 -4323.034,E2 -4323.034} C_VEL
LIN {X 0,Y 531.075,Z 222.33,A -85,B 0,C 180,E1 -4326.077,E2 -4326.077} C_VEL
LIN {X 0,Y 531.017,Z 222.339,A -85,B 0,C 180,E1 -4329.138,E2 -4329.138} C_VEL
LIN {X 0,Y 531.028,Z 222.339,A -85,B 0,C 180,E1 -4332.225,E2 -4332.225} C_VEL
LIN {X 0,Y 530.986,Z 222.345,A -85,B 0,C 180,E1 -4335.35,E2 -4335.35} C_VEL
LIN {X 0,Y 531.006,Z 222.338,A -85,B 0,C 180,E1 -4337.723,E2 -4337.723} C_VEL
LIN {X 0,Y 530.988,Z 222.341,A -85,B 0,C 180,E1 -4340.938,E2 -4340.938} C_VEL
LIN {X 0,Y 530.953,Z 222.345,A -85,B 0,C 180,E1 -4344.226,E2 -4344.226} C_VEL
LIN {X 0,Y 531.003,Z 222.344,A -85,B 0,C 180,E1 -4346.744,E2 -4346.744} C_VEL
LIN {X 0,Y 530.991,Z 222.34,A -85,B 0,C 180,E1 -4349.322,E2 -4349.322} C_VEL
LIN {X 0,Y 530.954,Z 222.348,A -85,B 0,C 180,E1 -4352.101,E2 -4352.101} C_VEL
LIN {X 0,Y 530.961,Z 222.348,A -85,B 0,C 180,E1 -4354.852,E2 -4354.852} C_VEL
LIN {X 0,Y 530.957,Z 222.344,A -85,B 0,C 180,E1 -4357.509,E2 -4357.509} C_VEL
LIN {X 0,Y 530.976,Z 222.344,A -85,B 0,C 180,E1 -4360.434,E2 -4360.434} C_VEL
LIN {X 0,Y 530.936,Z 222.352,A -85,B 0,C 180,E1 -4363.498,E2 -4363.498} C_VEL
LIN {X 0,Y 530.958,Z 222.35,A -85,B 0,C 180,E1 -4366.507,E2 -4366.507} C_VEL
LIN {X 0,Y 531.021,Z 222.342,A -85,B 0,C 180,E1 -4369.573,E2 -4369.573} C_VEL
LIN {X 0,Y 531.006,Z 222.489,A -85,B 0,C 180,E1 -4371.837,E2 -4371.837} C_VEL
LIN {X 0,Y 531.969,Z 228.522,A -85,B 0,C 180,E1 -4374.091,E2 -4374.091} C_VEL
LIN {X 0,Y 531.976,Z 235.036,A -85,B 0,C 180,E1 -4376.336,E2 -4376.336} C_VEL
LIN {X 0,Y 531.765,Z 242.998,A -85,B 0,C 180,E1 -4378.975,E2 -4378.975} C_VEL
LIN {X 0,Y 531.579,Z 252.372,A -85,B 0,C 180,E1 -4382.01,E2 -4382.01} C_VEL
LIN {X 0,Y 531.335,Z 261.638,A -85,B 0,C 180,E1 -4384.96,E2 -4384.96} C_VEL
LIN {X 0,Y 531.159,Z 270.915,A -85,B 0,C 180,E1 -4387.851,E2 -4387.851} C_VEL
LIN {X 0,Y 530.962,Z 280.173,A -85,B 0,C 180,E1 -4390.677,E2 -4390.677} C_VEL
LIN {X 0,Y 530.82,Z 289.44,A -85,B 0,C 180,E1 -4393.463,E2 -4393.463} C_VEL
LIN {X 0,Y 530.693,Z 299.534,A -85,B 0,C 180,E1 -4396.455,E2 -4396.455} C_VEL
LIN {X 0,Y 532.347,Z 310.399,A -85,B 0,C 180,E1 -4396.74,E2 -4396.74} C_VEL
LIN {X 0,Y 532.163,Z 322.508,A -85,B 0,C 180,E1 -4397.124,E2 -4397.124} C_VEL
LIN {X 0,Y 531.918,Z 333.513,A -85,B 0,C 180,E1 -4397.603,E2 -4397.603} C_VEL
LIN {X 0,Y 531.617,Z 345.454,A -85,B 0,C 180,E1 -4398.281,E2 -4398.281} C_VEL
LIN {X 0,Y 531.396,Z 357.113,A -85,B 0,C 180,E1 -4399.138,E2 -4399.138} C_VEL
LIN {X 0,Y 531.117,Z 367.55,A -85,B 0,C 180,E1 -4400.096,E2 -4400.096} C_VEL
LIN {X 0,Y 530.93,Z 376,A -85,B 0,C 180,E1 -4401.053,E2 -4401.053} C_VEL
LIN {X 0,Y 530.757,Z 384.245,A -85,B 0,C 180,E1 -4402.201,E2 -4402.201} C_VEL
LIN {X 0,Y 530.597,Z 391.275,A -85,B 0,C 180,E1 -4403.42,E2 -4403.42} C_VEL
LIN {X 0,Y 530.524,Z 396.954,A -85,B 0,C 180,E1 -4404.68,E2 -4404.68} C_VEL
LIN {X 0,Y 530.522,Z 400.898,A -85,B 0,C 180,E1 -4405.823,E2 -4405.823} C_VEL
LIN {X 0,Y 530.457,Z 403.81,A -85,B 0,C 180,E1 -4406.963,E2 -4406.963} C_VEL
LIN {X 0,Y 530.411,Z 405.199,A -85,B 0,C 180,E1 -4407.723,E2 -4407.723} C_VEL
LIN {X 0,Y 530.344,Z 406.786,A -85,B 0,C 180,E1 -4409.242,E2 -4409.242} C_VEL
LIN {X 0,Y 530.342,Z 407,A -85,B 0,C 180,E1 -4410.001,E2 -4410.001} C_VEL
LIN {X 0,Y 530.361,Z 406.185,A -85,B 0,C 180,E1 -4411.52,E2 -4411.52} C_VEL
LIN {X 0,Y 530.411,Z 405.197,A -85,B 0,C 180,E1 -4412.279,E2 -4412.279} C_VEL
LIN {X 0,Y 530.457,Z 403.808,A -85,B 0,C 180,E1 -4413.039,E2 -4413.039} C_VEL
LIN {X 0,Y 530.523,Z 400.893,A -85,B 0,C 180,E1 -4414.179,E2 -4414.179} C_VEL
LIN {X 0,Y 530.525,Z 396.945,A -85,B 0,C 180,E1 -4415.322,E2 -4415.322} C_VEL
LIN {X 0,Y 530.6,Z 391.257,A -85,B 0,C 180,E1 -4416.583,E2 -4416.583} C_VEL
LIN {X 0,Y 530.759,Z 384.23,A -85,B 0,C 180,E1 -4417.802,E2 -4417.802} C_VEL
LIN {X 0,Y 530.93,Z 375.982,A -85,B 0,C 180,E1 -4418.949,E2 -4418.949} C_VEL
LIN {X 0,Y 531.119,Z 367.528,A -85,B 0,C 180,E1 -4419.906,E2 -4419.906} C_VEL
LIN {X 0,Y 531.394,Z 357.085,A -85,B 0,C 180,E1 -4420.864,E2 -4420.864} C_VEL
LIN {X 0,Y 531.636,Z 346.431,A -85,B 0,C 180,E1 -4421.652,E2 -4421.652} C_VEL
LIN {X 0,Y 531.856,Z 335.39,A -85,B 0,C 180,E1 -4422.304,E2 -4422.304} C_VEL
LIN {X 0,Y 532.091,Z 323.735,A -85,B 0,C 180,E1 -4422.831,E2 -4422.831} C_VEL
LIN {X 0,Y 532.32,Z 310.308,A -85,B 0,C 180,E1 -4423.262,E2 -4423.262} C_VEL
LIN {X 0,Y 530.69,Z 299.527,A -85,B 0,C 180,E1 -4423.548,E2 -4423.548} C_VEL
LIN {X 0,Y 530.814,Z 290.756,A -85,B 0,C 180,E1 -4426.144,E2 -4426.144} C_VEL
LIN {X 0,Y 530.958,Z 281.489,A -85,B 0,C 180,E1 -4428.924,E2 -4428.924} C_VEL
LIN {X 0,Y 531.12,Z 272.221,A -85,B 0,C 180,E1 -4431.748,E2 -4431.748} C_VEL
LIN {X 0,Y 531.335,Z 262.954,A -85,B 0,C 180,E1 -4434.624,E2 -4434.624} C_VEL
LIN {X 0,Y 531.542,Z 253.457,A -85,B 0,C 180,E1 -4437.641,E2 -4437.641} C_VEL
LIN {X 0,Y 531.798,Z 243.097,A -85,B 0,C 180,E1 -4441.026,E2 -4441.026} C_VEL
LIN {X 0,Y 531.986,Z 234.892,A -85,B 0,C 180,E1 -4443.702,E2 -4443.702} C_VEL
LIN {X 0,Y 531.99,Z 228.526,A -85,B 0,C 180,E1 -4445.911,E2 -4445.911} C_VEL
LIN {X 0,Y 530.975,Z 222.348,A -85,B 0,C 180,E1 -4448.228,E2 -4448.228} C_VEL
LIN {X 0,Y 530.99,Z 222.342,A -85,B 0,C 180,E1 -4451.437,E2 -4451.437} C_VEL
LIN {X 0,Y 530.992,Z 222.343,A -85,B 0,C 180,E1 -4454.548,E2 -4454.548} C_VEL
LIN {X 0,Y 530.988,Z 222.345,A -85,B 0,C 180,E1 -4457.835,E2 -4457.835} C_VEL
LIN {X 0,Y 530.977,Z 222.343,A -85,B 0,C 180,E1 -4460.556,E2 -4460.556} C_VEL
LIN {X 0,Y 530.95,Z 222.346,A -85,B 0,C 180,E1 -4463.441,E2 -4463.441} C_VEL
LIN {X 0,Y 530.966,Z 222.349,A -85,B 0,C 180,E1 -4466.501,E2 -4466.501} C_VEL
LIN {X 0,Y 530.964,Z 222.344,A -85,B 0,C 180,E1 -4469.358,E2 -4469.358} C_VEL
LIN {X 0,Y 530.972,Z 222.346,A -85,B 0,C 180,E1 -4471.543,E2 -4471.543} C_VEL
LIN {X 0,Y 530.991,Z 222.341,A -85,B 0,C 180,E1 -4474.163,E2 -4474.163} C_VEL
LIN {X 0,Y 530.96,Z 222.346,A -85,B 0,C 180,E1 -4476.603,E2 -4476.603} C_VEL
LIN {X 0,Y 531.005,Z 222.342,A -85,B 0,C 180,E1 -4479.062,E2 -4479.062} C_VEL
LIN {X 0,Y 530.975,Z 222.342,A -85,B 0,C 180,E1 -4481.478,E2 -4481.478} C_VEL
LIN {X 0,Y 531.025,Z 222.335,A -85,B 0,C 180,E1 -4485.05,E2 -4485.05} C_VEL
LIN {X 0,Y 531.016,Z 222.337,A -85,B 0,C 180,E1 -4488.351,E2 -4488.351} C_VEL
LIN {X 0,Y 531.035,Z 222.338,A -85,B 0,C 180,E1 -4491.629,E2 -4491.629} C_VEL
LIN {X 0,Y 531.079,Z 222.329,A -85,B 0,C 180,E1 -4493.923,E2 -4493.923} C_VEL
LIN {X 0,Y 531.11,Z 222.329,A -85,B 0,C 180,E1 -4496.966,E2 -4496.966} C_VEL
LIN {X 0,Y 531.151,Z 222.326,A -85,B 0,C 180,E1 -4500,E2 -4500} C_VEL
LIN {X 0,Y 531.099,Z 222.327,A -85,B 0,C 180,E1 -4503.034,E2 -4503.034} C_VEL
LIN {X 0,Y 531.037,Z 222.334,A -85,B 0,C 180,E1 -4506.078,E2 -4506.078} C_VEL
LIN {X 0,Y 531.011,Z 222.343,A -85,B 0,C 180,E1 -4509.139,E2 -4509.139} C_VEL
LIN {X 0,Y 531.035,Z 222.338,A -85,B 0,C 180,E1 -4512.225,E2 -4512.225} C_VEL
LIN {X 0,Y 531.002,Z 222.339,A -85,B 0,C 180,E1 -4515.35,E2 -4515.35} C_VEL
LIN {X 0,Y 530.993,Z 222.341,A -85,B 0,C 180,E1 -4518.521,E2 -4518.521} C_VEL
LIN {X 0,Y 531.006,Z 222.34,A -85,B 0,C 180,E1 -4520.938,E2 -4520.938} C_VEL
LIN {X 0,Y 530.952,Z 222.345,A -85,B 0,C 180,E1 -4524.226,E2 -4524.226} C_VEL
LIN {X 0,Y 530.961,Z 222.343,A -85,B 0,C 180,E1 -4527.52,E2 -4527.52} C_VEL
LIN {X 0,Y 530.957,Z 222.349,A -85,B 0,C 180,E1 -4530.198,E2 -4530.198} C_VEL
LIN {X 0,Y 530.974,Z 222.342,A -85,B 0,C 180,E1 -4532.866,E2 -4532.866} C_VEL
LIN {X 0,Y 530.958,Z 222.349,A -85,B 0,C 180,E1 -4535.62,E2 -4535.62} C_VEL
LIN {X 0,Y 530.971,Z 222.344,A -85,B 0,C 180,E1 -4538.653,E2 -4538.653} C_VEL
LIN {X 0,Y 530.987,Z 222.342,A -85,B 0,C 180,E1 -4541.437,E2 -4541.437} C_VEL
LIN {X 0,Y 530.944,Z 222.346,A -85,B 0,C 180,E1 -4543.513,E2 -4543.513} C_VEL
LIN {X 0,Y 530.272,Z 222.434,A -85,B 0,C 180,E1 -4544.146,E2 -4544.146} C_VEL
LIN {X 0,Y 527.426,Z 222.786,A -85,B 0,C 180,E1 -4545.175,E2 -4545.175} C_VEL
LIN {X 0,Y 525.016,Z 223.088,A -85,B 0,C 180,E1 -4546.003,E2 -4546.003} C_VEL
LIN {X 0,Y 523.968,Z 223.217,A -85,B 0,C 180,E1 -4546.643,E2 -4546.643} C_VEL
LIN {X 0,Y 523.876,Z 223.226,A -85,B 0,C 180,E1 -4546.859,E2 -4546.859} C_VEL
LIN {X 0,Y 523.904,Z 223.229,A -85,B 0,C 180,E1 -4549.915,E2 -4549.915} C_VEL
LIN {X 0,Y 523.912,Z 223.224,A -85,B 0,C 180,E1 -4552.867,E2 -4552.867} C_VEL
LIN {X 0,Y 523.927,Z 223.222,A -85,B 0,C 180,E1 -4555.708,E2 -4555.708} C_VEL
LIN {X 0,Y 523.884,Z 223.23,A -85,B 0,C 180,E1 -4558.452,E2 -4558.452} C_VEL
LIN {X 0,Y 523.624,Z 223.264,A -85,B 0,C 180,E1 -4560.742,E2 -4560.742} C_VEL
LIN {X 0,Y 523.581,Z 225.534,A -85,B 0,C 180,E1 -4562.845,E2 -4562.845} C_VEL
LIN {X 0,Y 523.589,Z 228.863,A -85,B 0,C 180,E1 -4565.889,E2 -4565.889} C_VEL
LIN {X 0,Y 523.492,Z 232.012,A -85,B 0,C 180,E1 -4568.746,E2 -4568.746} C_VEL
LIN {X 0,Y 523.466,Z 234.735,A -85,B 0,C 180,E1 -4571.202,E2 -4571.202} C_VEL
LIN {X 0,Y 523.466,Z 237.455,A -85,B 0,C 180,E1 -4573.623,E2 -4573.623} C_VEL
LIN {X 0,Y 523.457,Z 240.198,A -85,B 0,C 180,E1 -4576.014,E2 -4576.014} C_VEL
LIN {X 0,Y 523.495,Z 243.068,A -85,B 0,C 180,E1 -4578.534,E2 -4578.534} C_VEL
LIN {X 0,Y 523.404,Z 245.293,A -85,B 0,C 180,E1 -4580.385,E2 -4580.385} C_VEL
LIN {X 0,Y 525.419,Z 255.703,A -85,B 0,C 180,E1 -4580.714,E2 -4580.714} C_VEL
LIN {X 0,Y 525.21,Z 268.778,A -85,B 0,C 180,E1 -4581.195,E2 -4581.195} C_VEL
LIN {X 0,Y 524.99,Z 281.167,A -85,B 0,C 180,E1 -4581.822,E2 -4581.822} C_VEL
LIN {X 0,Y 524.656,Z 292.127,A -85,B 0,C 180,E1 -4582.543,E2 -4582.543} C_VEL
LIN {X 0,Y 524.444,Z 303.141,A -85,B 0,C 180,E1 -4583.458,E2 -4583.458} C_VEL
LIN {X 0,Y 524.139,Z 312.526,A -85,B 0,C 180,E1 -4584.42,E2 -4584.42} C_VEL
LIN {X 0,Y 523.858,Z 321.561,A -85,B 0,C 180,E1 -4585.575,E2 -4585.575} C_VEL
LIN {X 0,Y 523.686,Z 328.831,A -85,B 0,C 180,E1 -4586.729,E2 -4586.729} C_VEL
LIN {X 0,Y 523.536,Z 335.539,A -85,B 0,C 180,E1 -4588.076,E2 -4588.076} C_VEL
LIN {X 0,Y 523.34,Z 339.978,A -85,B 0,C 180,E1 -4589.229,E2 -4589.229} C_VEL
LIN {X 0,Y 523.325,Z 342.314,A -85,B 0,C 180,E1 -4589.999,E2 -4589.999} C_VEL
LIN {X 0,Y 523.287,Z 344.233,A -85,B 0,C 180,E1 -4590.768,E2 -4590.768} C_VEL
LIN {X 0,Y 523.288,Z 345.744,A -85,B 0,C 180,E1 -4591.538,E2 -4591.538} C_VEL
LIN {X 0,Y 523.415,Z 347.482,A -85,B 0,C 180,E1 -4593.078,E2 -4593.078} C_VEL
LIN {X 0,Y 523.4,Z 347.783,A -85,B 0,C 180,E1 -4593.848,E2 -4593.848} C_VEL
LIN {X 0,Y 523.318,Z 347.711,A -85,B 0,C 180,E1 -4594.621,E2 -4594.621} C_VEL
LIN {X 0,Y 523.37,Z 347.209,A -85,B 0,C 180,E1 -4595.393,E2 -4595.393} C_VEL
LIN {X 0,Y 523.383,Z 345.018,A -85,B 0,C 180,E1 -4596.94,E2 -4596.94} C_VEL
LIN {X 0,Y 523.425,Z 342.277,A -85,B 0,C 180,E1 -4598.104,E2 -4598.104} C_VEL
LIN {X 0,Y 523.469,Z 338.511,A -85,B 0,C 180,E1 -4599.27,E2 -4599.27} C_VEL
LIN {X 0,Y 523.569,Z 333.608,A -85,B 0,C 180,E1 -4600.439,E2 -4600.439} C_VEL
LIN {X 0,Y 523.764,Z 327.414,A -85,B 0,C 180,E1 -4601.61,E2 -4601.61} C_VEL
LIN {X 0,Y 523.948,Z 319.639,A -85,B 0,C 180,E1 -4602.786,E2 -4602.786} C_VEL
LIN {X 0,Y 524.138,Z 311.658,A -85,B 0,C 180,E1 -4603.767,E2 -4603.767} C_VEL
LIN {X 0,Y 524.43,Z 301.882,A -85,B 0,C 180,E1 -4604.75,E2 -4604.75} C_VEL
LIN {X 0,Y 524.676,Z 290.938,A -85,B 0,C 180,E1 -4605.638,E2 -4605.638} C_VEL
LIN {X 0,Y 524.964,Z 280.158,A -85,B 0,C 180,E1 -4606.327,E2 -4606.327} C_VEL
LIN {X 0,Y 525.208,Z 267.107,A -85,B 0,C 180,E1 -4606.969,E2 -4606.969} C_VEL
LIN {X 0,Y 525.359,Z 254.961,A -85,B 0,C 180,E1 -4607.402,E2 -4607.402} C_VEL
LIN {X 0,Y 523.415,Z 245.229,A -85,B 0,C 180,E1 -4607.702,E2 -4607.702} C_VEL
LIN {X 0,Y 523.379,Z 242.102,A -85,B 0,C 180,E1 -4610.433,E2 -4610.433} C_VEL
LIN {X 0,Y 523.42,Z 239.263,A -85,B 0,C 180,E1 -4612.915,E2 -4612.915} C_VEL
LIN {X 0,Y 523.523,Z 235.865,A -85,B 0,C 180,E1 -4615.915,E2 -4615.915} C_VEL
LIN {X 0,Y 523.553,Z 232.574,A -85,B 0,C 180,E1 -4618.896,E2 -4618.896} C_VEL
LIN {X 0,Y 523.561,Z 229.689,A -85,B 0,C 180,E1 -4621.567,E2 -4621.567} C_VEL
LIN {X 0,Y 523.638,Z 226.748,A -85,B 0,C 180,E1 -4624.311,E2 -4624.311} C_VEL
LIN {X 0,Y 523.665,Z 223.707,A -85,B 0,C 180,E1 -4627.151,E2 -4627.151} C_VEL
LIN {X 0,Y 523.67,Z 223.258,A -85,B 0,C 180,E1 -4627.644,E2 -4627.644} C_VEL
LIN {X 0,Y 523.906,Z 223.223,A -85,B 0,C 180,E1 -4630.125,E2 -4630.125} C_VEL
LIN {X 0,Y 523.932,Z 223.223,A -85,B 0,C 180,E1 -4632.458,E2 -4632.458} C_VEL
LIN {X 0,Y 523.947,Z 223.218,A -85,B 0,C 180,E1 -4635.308,E2 -4635.308} C_VEL
LIN {X 0,Y 523.943,Z 223.219,A -85,B 0,C 180,E1 -4638.689,E2 -4638.689} C_VEL
LIN {X 0,Y 523.91,Z 223.227,A -85,B 0,C 180,E1 -4641.079,E2 -4641.079} C_VEL
LIN {X 0,Y 523.92,Z 223.222,A -85,B 0,C 180,E1 -4643.827,E2 -4643.827} C_VEL
LIN {X 0,Y 523.905,Z 223.223,A -85,B 0,C 180,E1 -4646.633,E2 -4646.633} C_VEL
LIN {X 0,Y 523.939,Z 223.223,A -85,B 0,C 180,E1 -4649.354,E2 -4649.354} C_VEL
LIN {X 0,Y 523.971,Z 223.218,A -85,B 0,C 180,E1 -4652.28,E2 -4652.28} C_VEL
LIN {X 0,Y 523.946,Z 223.219,A -85,B 0,C 180,E1 -4654.581,E2 -4654.581} C_VEL
LIN {X 0,Y 523.906,Z 223.226,A -85,B 0,C 180,E1 -4657.106,E2 -4657.106} C_VEL
LIN {X 0,Y 523.968,Z 223.215,A -85,B 0,C 180,E1 -4659.865,E2 -4659.865} C_VEL
LIN {X 0,Y 523.957,Z 223.218,A -85,B 0,C 180,E1 -4662.837,E2 -4662.837} C_VEL
LIN {X 0,Y 523.966,Z 223.217,A -85,B 0,C 180,E1 -4665.235,E2 -4665.235} C_VEL
LIN {X 0,Y 524.001,Z 223.212,A -85,B 0,C 180,E1 -4668.394,E2 -4668.394} C_VEL
LIN {X 0,Y 523.988,Z 223.213,A -85,B 0,C 180,E1 -4671.516,E2 -4671.516} C_VEL
LIN {X 0,Y 524.095,Z 223.2,A -85,B 0,C 180,E1 -4674.614,E2 -4674.614} C_VEL
LIN {X 0,Y 524.098,Z 223.2,A -85,B 0,C 180,E1 -4677.694,E2 -4677.694} C_VEL
LIN {X 0,Y 524.109,Z 223.201,A -85,B 0,C 180,E1 -4680.768,E2 -4680.768} C_VEL
LIN {X 0,Y 524.062,Z 223.204,A -85,B 0,C 180,E1 -4683.075,E2 -4683.075} C_VEL
LIN {X 0,Y 524.037,Z 223.206,A -85,B 0,C 180,E1 -4686.159,E2 -4686.159} C_VEL
LIN {X 0,Y 523.985,Z 223.214,A -85,B 0,C 180,E1 -4689.262,E2 -4689.262} C_VEL
LIN {X 0,Y 523.99,Z 223.215,A -85,B 0,C 180,E1 -4691.739,E2 -4691.739} C_VEL
LIN {X 0,Y 523.981,Z 223.216,A -85,B 0,C 180,E1 -4695.053,E2 -4695.053} C_VEL
LIN {X 0,Y 523.954,Z 223.217,A -85,B 0,C 180,E1 -4697.969,E2 -4697.969} C_VEL
LIN {X 0,Y 523.96,Z 223.22,A -85,B 0,C 180,E1 -4700.411,E2 -4700.411} C_VEL
LIN {X 0,Y 523.897,Z 223.224,A -85,B 0,C 180,E1 -4702.894,E2 -4702.894} C_VEL
LIN {X 0,Y 523.976,Z 223.214,A -85,B 0,C 180,E1 -4706.021,E2 -4706.021} C_VEL
LIN {X 0,Y 523.942,Z 223.221,A -85,B 0,C 180,E1 -4708.875,E2 -4708.875} C_VEL
LIN {X 0,Y 523.912,Z 223.226,A -85,B 0,C 180,E1 -4711.545,E2 -4711.545} C_VEL
LIN {X 0,Y 523.923,Z 223.221,A -85,B 0,C 180,E1 -4714.291,E2 -4714.291} C_VEL
LIN {X 0,Y 523.898,Z 223.225,A -85,B 0,C 180,E1 -4717.133,E2 -4717.133} C_VEL
LIN {X 0,Y 523.929,Z 223.225,A -85,B 0,C 180,E1 -4720.131,E2 -4720.131} C_VEL
LIN {X 0,Y 523.915,Z 223.222,A -85,B 0,C 180,E1 -4722.459,E2 -4722.459} C_VEL
LIN {X 0,Y 523.947,Z 223.222,A -85,B 0,C 180,E1 -4725.31,E2 -4725.31} C_VEL
LIN {X 0,Y 523.967,Z 223.22,A -85,B 0,C 180,E1 -4728.689,E2 -4728.689} C_VEL
LIN {X 0,Y 523.947,Z 223.389,A -85,B 0,C 180,E1 -4731.597,E2 -4731.597} C_VEL
LIN {X 0,Y 524.988,Z 229.503,A -85,B 0,C 180,E1 -4733.914,E2 -4733.914} C_VEL
LIN {X 0,Y 525.02,Z 235.679,A -85,B 0,C 180,E1 -4736.093,E2 -4736.093} C_VEL
LIN {X 0,Y 524.77,Z 244.261,A -85,B 0,C 180,E1 -4738.995,E2 -4738.995} C_VEL
LIN {X 0,Y 524.555,Z 254.078,A -85,B 0,C 180,E1 -4742.162,E2 -4742.162} C_VEL
LIN {X 0,Y 524.321,Z 262.962,A -85,B 0,C 180,E1 -4745.026,E2 -4745.026} C_VEL
LIN {X 0,Y 524.127,Z 272.229,A -85,B 0,C 180,E1 -4747.949,E2 -4747.949} C_VEL
LIN {X 0,Y 523.922,Z 281.496,A -85,B 0,C 180,E1 -4750.815,E2 -4750.815} C_VEL
LIN {X 0,Y 523.758,Z 290.764,A -85,B 0,C 180,E1 -4753.634,E2 -4753.634} C_VEL
LIN {X 0,Y 523.674,Z 299.807,A -85,B 0,C 180,E1 -4756.288,E2 -4756.288} C_VEL
LIN {X 0,Y 525.451,Z 311.314,A -85,B 0,C 180,E1 -4756.588,E2 -4756.588} C_VEL
LIN {X 0,Y 525.246,Z 322.508,A -85,B 0,C 180,E1 -4756.952,E2 -4756.952} C_VEL
LIN {X 0,Y 524.971,Z 333.514,A -85,B 0,C 180,E1 -4757.436,E2 -4757.436} C_VEL
LIN {X 0,Y 524.669,Z 345.026,A -85,B 0,C 180,E1 -4758.095,E2 -4758.095} C_VEL
LIN {X 0,Y 524.457,Z 355.938,A -85,B 0,C 180,E1 -4758.895,E2 -4758.895} C_VEL
LIN {X 0,Y 524.21,Z 365.613,A -85,B 0,C 180,E1 -4759.769,E2 -4759.769} C_VEL
LIN {X 0,Y 523.928,Z 374.423,A -85,B 0,C 180,E1 -4760.738,E2 -4760.738} C_VEL
LIN {X 0,Y 523.722,Z 383.009,A -85,B 0,C 180,E1 -4761.901,E2 -4761.901} C_VEL
LIN {X 0,Y 523.573,Z 389.874,A -85,B 0,C 180,E1 -4763.062,E2 -4763.062} C_VEL
LIN {X 0,Y 523.543,Z 395.371,A -85,B 0,C 180,E1 -4764.223,E2 -4764.223} C_VEL
LIN {X 0,Y 523.36,Z 399.681,A -85,B 0,C 180,E1 -4765.38,E2 -4765.38} C_VEL
LIN {X 0,Y 523.443,Z 401.961,A -85,B 0,C 180,E1 -4766.152,E2 -4766.152} C_VEL
LIN {X 0,Y 523.367,Z 403.81,A -85,B 0,C 180,E1 -4766.922,E2 -4766.922} C_VEL
LIN {X 0,Y 523.335,Z 405.199,A -85,B 0,C 180,E1 -4767.692,E2 -4767.692} C_VEL
LIN {X 0,Y 523.25,Z 406.786,A -85,B 0,C 180,E1 -4769.232,E2 -4769.232} C_VEL
LIN {X 0,Y 523.246,Z 407,A -85,B 0,C 180,E1 -4770.001,E2 -4770.001} C_VEL
LIN {X 0,Y 523.275,Z 406.185,A -85,B 0,C 180,E1 -4771.54,E2 -4771.54} C_VEL
LIN {X 0,Y 523.335,Z 405.197,A -85,B 0,C 180,E1 -4772.31,E2 -4772.31} C_VEL
LIN {X 0,Y 523.368,Z 403.808,A -85,B 0,C 180,E1 -4773.08,E2 -4773.08} C_VEL
LIN {X 0,Y 523.442,Z 400.893,A -85,B 0,C 180,E1 -4774.236,E2 -4774.236} C_VEL
LIN {X 0,Y 523.464,Z 396.945,A -85,B 0,C 180,E1 -4775.394,E2 -4775.394} C_VEL
LIN {X 0,Y 523.525,Z 391.72,A -85,B 0,C 180,E1 -4776.582,E2 -4776.582} C_VEL
LIN {X 0,Y 523.666,Z 385.461,A -85,B 0,C 180,E1 -4777.714,E2 -4777.714} C_VEL
LIN {X 0,Y 523.856,Z 377.47,A -85,B 0,C 180,E1 -4778.876,E2 -4778.876} C_VEL
LIN {X 0,Y 524.06,Z 369.325,A -85,B 0,C 180,E1 -4779.846,E2 -4779.846} C_VEL
LIN {X 0,Y 524.336,Z 359.388,A -85,B 0,C 180,E1 -4780.817,E2 -4780.817} C_VEL
LIN {X 0,Y 524.631,Z 348.218,A -85,B 0,C 180,E1 -4781.687,E2 -4781.687} C_VEL
LIN {X 0,Y 524.846,Z 337.157,A -85,B 0,C 180,E1 -4782.373,E2 -4782.373} C_VEL
LIN {X 0,Y 525.152,Z 324.954,A -85,B 0,C 180,E1 -4782.955,E2 -4782.955} C_VEL
LIN {X 0,Y 525.38,Z 312.136,A -85,B 0,C 180,E1 -4783.392,E2 -4783.392} C_VEL
LIN {X 0,Y 524.747,Z 306.317,A -85,B 0,C 180,E1 -4783.556,E2 -4783.556} C_VEL
LIN {X 0,Y 523.628,Z 299.527,A -85,B 0,C 180,E1 -4783.734,E2 -4783.734} C_VEL
LIN {X 0,Y 523.762,Z 290.756,A -85,B 0,C 180,E1 -4786.368,E2 -4786.368} C_VEL
LIN {X 0,Y 523.926,Z 281.489,A -85,B 0,C 180,E1 -4789.188,E2 -4789.188} C_VEL
LIN {X 0,Y 524.132,Z 271.434,A -85,B 0,C 180,E1 -4792.3,E2 -4792.3} C_VEL
LIN {X 0,Y 524.353,Z 261.63,A -85,B 0,C 180,E1 -4795.399,E2 -4795.399} C_VEL
LIN {X 0,Y 524.612,Z 252.363,A -85,B 0,C 180,E1 -4798.398,E2 -4798.398} C_VEL
LIN {X 0,Y 524.831,Z 242.906,A -85,B 0,C 180,E1 -4801.484,E2 -4801.484} C_VEL
LIN {X 0,Y 525.032,Z 234.746,A -85,B 0,C 180,E1 -4804.21,E2 -4804.21} C_VEL
LIN {X 0,Y 525.009,Z 229.511,A -85,B 0,C 180,E1 -4806.087,E2 -4806.087} C_VEL
LIN {X 0,Y 523.913,Z 223.228,A -85,B 0,C 180,E1 -4808.532,E2 -4808.532} C_VEL
LIN {X 0,Y 523.949,Z 223.22,A -85,B 0,C 180,E1 -4811.309,E2 -4811.309} C_VEL
LIN {X 0,Y 523.961,Z 223.218,A -85,B 0,C 180,E1 -4814.692,E2 -4814.692} C_VEL
LIN {X 0,Y 523.958,Z 223.22,A -85,B 0,C 180,E1 -4817.881,E2 -4817.881} C_VEL
LIN {X 0,Y 523.919,Z 223.226,A -85,B 0,C 180,E1 -4820.915,E2 -4820.915} C_VEL
LIN {X 0,Y 523.885,Z 223.225,A -85,B 0,C 180,E1 -4823.824,E2 -4823.824} C_VEL
LIN {X 0,Y 523.915,Z 223.226,A -85,B 0,C 180,E1 -4826.634,E2 -4826.634} C_VEL
LIN {X 0,Y 523.947,Z 223.218,A -85,B 0,C 180,E1 -4829.355,E2 -4829.355} C_VEL
LIN {X 0,Y 523.951,Z 223.219,A -85,B 0,C 180,E1 -4832.289,E2 -4832.289} C_VEL
LIN {X 0,Y 523.936,Z 223.22,A -85,B 0,C 180,E1 -4834.58,E2 -4834.58} C_VEL
LIN {X 0,Y 523.917,Z 223.226,A -85,B 0,C 180,E1 -4837.107,E2 -4837.107} C_VEL
LIN {X 0,Y 523.986,Z 223.213,A -85,B 0,C 180,E1 -4839.866,E2 -4839.866} C_VEL
LIN {X 0,Y 523.925,Z 223.222,A -85,B 0,C 180,E1 -4842.836,E2 -4842.836} C_VEL
LIN {X 0,Y 523.967,Z 223.214,A -85,B 0,C 180,E1 -4845.235,E2 -4845.235} C_VEL
LIN {X 0,Y 523.964,Z 223.215,A -85,B 0,C 180,E1 -4848.393,E2 -4848.393} C_VEL
LIN {X 0,Y 523.987,Z 223.217,A -85,B 0,C 180,E1 -4851.516,E2 -4851.516} C_VEL
LIN {X 0,Y 524.041,Z 223.206,A -85,B 0,C 180,E1 -4853.841,E2 -4853.841} C_VEL
LIN {X 0,Y 524.076,Z 223.205,A -85,B 0,C 180,E1 -4856.925,E2 -4856.925} C_VEL
LIN {X 0,Y 524.122,Z 223.202,A -85,B 0,C 180,E1 -4860,E2 -4860} C_VEL
LIN {X 0,Y 524.041,Z 223.206,A -85,B 0,C 180,E1 -4863.075,E2 -4863.075} C_VEL
LIN {X 0,Y 524.001,Z 223.21,A -85,B 0,C 180,E1 -4866.16,E2 -4866.16} C_VEL
LIN {X 0,Y 523.982,Z 223.217,A -85,B 0,C 180,E1 -4869.262,E2 -4869.262} C_VEL
LIN {X 0,Y 524.004,Z 223.211,A -85,B 0,C 180,E1 -4871.736,E2 -4871.736} C_VEL
LIN {X 0,Y 524.001,Z 223.212,A -85,B 0,C 180,E1 -4875.052,E2 -4875.052} C_VEL
LIN {X 0,Y 523.955,Z 223.221,A -85,B 0,C 180,E1 -4877.969,E2 -4877.969} C_VEL
LIN {X 0,Y 523.965,Z 223.216,A -85,B 0,C 180,E1 -4880.411,E2 -4880.411} C_VEL
LIN {X 0,Y 523.913,Z 223.225,A -85,B 0,C 180,E1 -4882.894,E2 -4882.894} C_VEL
LIN {X 0,Y 523.876,Z 223.227,A -85,B 0,C 180,E1 -4885.423,E2 -4885.423} C_VEL
LIN {X 0,Y 523.907,Z 223.223,A -85,B 0,C 180,E1 -4888.003,E2 -4888.003} C_VEL
LIN {X 0,Y 523.942,Z 223.219,A -85,B 0,C 180,E1 -4890.853,E2 -4890.853} C_VEL
LIN {X 0,Y 523.938,Z 223.223,A -85,B 0,C 180,E1 -4893.729,E2 -4893.729} C_VEL
LIN {X 0,Y 523.906,Z 223.223,A -85,B 0,C 180,E1 -4896.4,E2 -4896.4} C_VEL
LIN {X 0,Y 523.926,Z 223.225,A -85,B 0,C 180,E1 -4899.085,E2 -4899.085} C_VEL
LIN {X 0,Y 523.945,Z 223.219,A -85,B 0,C 180,E1 -4902.12,E2 -4902.12} C_VEL
LIN {X 0,Y 523.938,Z 223.218,A -85,B 0,C 180,E1 -4905.311,E2 -4905.311} C_VEL
LIN {X 0,Y 523.876,Z 223.226,A -85,B 0,C 180,E1 -4906.859,E2 -4906.859} C_VEL
LIN {X 0,Y 523.185,Z 223.313,A -85,B 0,C 180,E1 -4907.501,E2 -4907.501} C_VEL
LIN {X 0,Y 520.313,Z 223.671,A -85,B 0,C 180,E1 -4908.542,E2 -4908.542} C_VEL
LIN {X 0,Y 517.918,Z 223.97,A -85,B 0,C 180,E1 -4909.381,E2 -4909.381} C_VEL
LIN {X 0,Y 516.919,Z 224.097,A -85,B 0,C 180,E1 -4910.028,E2 -4910.028} C_VEL
LIN {X 0,Y 516.852,Z 224.103,A -85,B 0,C 180,E1 -4910.247,E2 -4910.247} C_VEL
